(* IEC 61131-3 sources: rust-plc/playground, 18 files *)

(* ---- 10_classes.st ---- *)
(*
 * Classes and OOP — IEC 61131-3 Object-Oriented Extensions
 *
 * Demonstrates the full OOP feature set:
 * - CLASS with VAR blocks, methods, and properties
 * - INTERFACE with method prototypes
 * - Inheritance via EXTENDS
 * - Interface implementation via IMPLEMENTS
 * - Access specifiers: PUBLIC, PRIVATE, PROTECTED
 * - ABSTRACT classes and methods
 * - FINAL classes and methods
 * - OVERRIDE for method overriding
 * - Properties with GET / SET accessors
 *
 * Run with: st-cli run playground/10_classes.st -n 10
 *)

// ═══════════════════════════════════════════════════════════════════════
// Interfaces — define contracts that classes must fulfill
// ═══════════════════════════════════════════════════════════════════════

INTERFACE IResettable
    METHOD Reset
    END_METHOD
END_INTERFACE

INTERFACE ICountable
    METHOD GetCount : INT
    END_METHOD
END_INTERFACE

// Interfaces can extend other interfaces
INTERFACE IFullCounter EXTENDS ICountable
    METHOD Increment
    END_METHOD
    METHOD Decrement
    END_METHOD
END_INTERFACE

// ═══════════════════════════════════════════════════════════════════════
// Basic class — encapsulates state + behavior
// ═══════════════════════════════════════════════════════════════════════

CLASS Counter IMPLEMENTS IFullCounter, IResettable
VAR
    _count : INT := 0;
    _maxCount : INT := 1000;
END_VAR

    // Public method — accessible from anywhere
    PUBLIC METHOD Increment
        IF _count < _maxCount THEN
            _count := _count + 1;
        END_IF;
    END_METHOD

    PUBLIC METHOD Decrement
        IF _count > 0 THEN
            _count := _count - 1;
        END_IF;
    END_METHOD

    PUBLIC METHOD GetCount : INT
        GetCount := _count;
    END_METHOD

    PUBLIC METHOD Reset
        _count := 0;
    END_METHOD

    // Private helper — only visible inside this class
    PRIVATE METHOD IsAtLimit : BOOL
    VAR
        result : BOOL;
    END_VAR
        result := (_count >= _maxCount);
        IsAtLimit := result;
    END_METHOD

    // Property — syntactic sugar for getter/setter
    PUBLIC PROPERTY Count : INT
        GET
            Count := _count;
        END_GET
        SET
            _count := Count;
        END_SET
    END_PROPERTY

    // Read-only property (getter only)
    PUBLIC PROPERTY MaxCount : INT
        GET
            MaxCount := _maxCount;
        END_GET
    END_PROPERTY
END_CLASS

// ═══════════════════════════════════════════════════════════════════════
// Inheritance — EXTENDS builds on existing classes
// ═══════════════════════════════════════════════════════════════════════

CLASS StepCounter EXTENDS Counter
VAR
    _stepSize : INT := 1;
    _accumulated : INT := 0;
END_VAR

    // Override changes the behavior of a parent method
    OVERRIDE METHOD Increment
    VAR
        i : INT;
    END_VAR
        _accumulated := _accumulated + _stepSize;
    END_METHOD

    PUBLIC METHOD SetStep
    VAR_INPUT
        step : INT;
    END_VAR
        IF step > 0 THEN
            _stepSize := step;
        END_IF;
    END_METHOD

    PUBLIC METHOD GetAccumulated : INT
        GetAccumulated := _accumulated;
    END_METHOD
END_CLASS

// ═══════════════════════════════════════════════════════════════════════
// Abstract classes — cannot be instantiated, define a template
// ═══════════════════════════════════════════════════════════════════════

ABSTRACT CLASS Shape
VAR
    _x : REAL := 0.0;
    _y : REAL := 0.0;
END_VAR

    // Abstract methods MUST be implemented by subclasses
    ABSTRACT METHOD Area : REAL
    END_METHOD

    ABSTRACT METHOD Perimeter : REAL
    END_METHOD

    // Concrete methods CAN be inherited as-is
    PUBLIC METHOD MoveTo
    VAR_INPUT
        newX : REAL;
        newY : REAL;
    END_VAR
        _x := newX;
        _y := newY;
    END_METHOD

    PUBLIC METHOD GetX : REAL
        GetX := _x;
    END_METHOD

    PUBLIC METHOD GetY : REAL
        GetY := _y;
    END_METHOD
END_CLASS

CLASS Rectangle EXTENDS Shape
VAR
    _width  : REAL := 0.0;
    _height : REAL := 0.0;
END_VAR

    PUBLIC METHOD SetSize
    VAR_INPUT
        w : REAL;
        h : REAL;
    END_VAR
        _width := w;
        _height := h;
    END_METHOD

    // Implementing the abstract methods
    OVERRIDE METHOD Area : REAL
        Area := _width * _height;
    END_METHOD

    OVERRIDE METHOD Perimeter : REAL
        Perimeter := 2.0 * (_width + _height);
    END_METHOD
END_CLASS

CLASS Circle EXTENDS Shape
VAR
    _radius : REAL := 0.0;
END_VAR

    PUBLIC METHOD SetRadius
    VAR_INPUT
        r : REAL;
    END_VAR
        _radius := r;
    END_METHOD

    OVERRIDE METHOD Area : REAL
        Area := 3.14159 * _radius * _radius;
    END_METHOD

    OVERRIDE METHOD Perimeter : REAL
        Perimeter := 2.0 * 3.14159 * _radius;
    END_METHOD
END_CLASS

// ═══════════════════════════════════════════════════════════════════════
// Final class — cannot be subclassed (sealed)
// ═══════════════════════════════════════════════════════════════════════

FINAL CLASS Logger
VAR
    _lastCode : INT := 0;
    _entryCount : INT := 0;
END_VAR

    PUBLIC METHOD Log
    VAR_INPUT
        code : INT;
    END_VAR
        _lastCode := code;
        _entryCount := _entryCount + 1;
    END_METHOD

    // Final method — cannot be overridden even if class is subclassed
    FINAL METHOD GetLastCode : INT
        GetLastCode := _lastCode;
    END_METHOD

    PUBLIC METHOD GetEntryCount : INT
        GetEntryCount := _entryCount;
    END_METHOD
END_CLASS

// ═══════════════════════════════════════════════════════════════════════
// Access specifiers — control visibility of members
// ═══════════════════════════════════════════════════════════════════════

CLASS AccessDemo
VAR
    _secret  : INT := 42;    // Only accessible within this class
    _shared  : INT := 0;     // Accessible within hierarchy
    _open    : INT := 0;     // Accessible from anywhere
END_VAR

    PRIVATE METHOD GetSecret : INT
        GetSecret := _secret;
    END_METHOD

    PROTECTED METHOD GetShared : INT
        GetShared := _shared;
    END_METHOD

    PUBLIC METHOD GetOpen : INT
        GetOpen := _open;
    END_METHOD

    PUBLIC METHOD SetAll
    VAR_INPUT
        val : INT;
    END_VAR
        _secret := val;
        _shared := val;
        _open := val;
    END_METHOD
END_CLASS

// ═══════════════════════════════════════════════════════════════════════
// Industrial example — PID controller as a class
// ═══════════════════════════════════════════════════════════════════════

CLASS PidController IMPLEMENTS IResettable
VAR_INPUT
    setpoint : REAL;
    feedback : REAL;
END_VAR
VAR_OUTPUT
    output : REAL;
END_VAR
VAR
    _kp : REAL := 1.0;
    _ki : REAL := 0.1;
    _kd : REAL := 0.01;
    _integral   : REAL := 0.0;
    _prevError  : REAL := 0.0;
    _outMin     : REAL := 0.0;
    _outMax     : REAL := 100.0;
END_VAR

    PUBLIC METHOD Configure
    VAR_INPUT
        kp : REAL;
        ki : REAL;
        kd : REAL;
        minOut : REAL;
        maxOut : REAL;
    END_VAR
        _kp := kp;
        _ki := ki;
        _kd := kd;
        _outMin := minOut;
        _outMax := maxOut;
    END_METHOD

    PUBLIC METHOD Execute
    VAR
        error : REAL;
        derivative : REAL;
        raw : REAL;
    END_VAR
        error := setpoint - feedback;
        _integral := _integral + error;
        derivative := error - _prevError;
        _prevError := error;

        raw := _kp * error + _ki * _integral + _kd * derivative;

        // Clamp output
        IF raw < _outMin THEN
            output := _outMin;
        ELSIF raw > _outMax THEN
            output := _outMax;
        ELSE
            output := raw;
        END_IF;
    END_METHOD

    PUBLIC METHOD Reset
        _integral := 0.0;
        _prevError := 0.0;
        output := 0.0;
    END_METHOD
END_CLASS

// ═══════════════════════════════════════════════════════════════════════
// Main program — ties it all together
// ═══════════════════════════════════════════════════════════════════════

VAR_GLOBAL
    g_counter_value : INT;
    g_step_counter_value : INT;
    g_rect_area : REAL;
    g_circle_area : REAL;
    g_pid_output : REAL;
    g_log_entries : INT;
END_VAR

PROGRAM Main
VAR
    // Class instances — just like FB instances
    cnt       : Counter;
    stepCnt   : StepCounter;
    rect      : Rectangle;
    circ      : Circle;
    pid       : PidController;
    logger    : Logger;
    access    : AccessDemo;

    cycle     : INT := 0;
    simTemp   : REAL := 20.0;
END_VAR
    cycle := cycle + 1;

    // ── Counter demo ──
    cnt.Increment();
    cnt.Increment();
    cnt.Increment();
    g_counter_value := cnt.GetCount();

    // ── Step counter (inherited + overridden) ──
    stepCnt.SetStep(step := 5);
    stepCnt.Increment();   // Accumulates 5 instead of 1
    g_step_counter_value := stepCnt.GetAccumulated();

    // ── Shapes (abstract base, concrete subclasses) ──
    rect.SetSize(w := 4.0, h := 3.0);
    rect.MoveTo(newX := 10.0, newY := 20.0);
    g_rect_area := rect.Area();          // 12.0

    circ.SetRadius(r := 5.0);
    g_circle_area := circ.Area();        // ~78.54

    // ── PID controller ──
    pid.Configure(kp := 2.0, ki := 0.5, kd := 0.1,
                  minOut := 0.0, maxOut := 100.0);
    pid.setpoint := 50.0;
    pid.feedback := simTemp;
    pid.Execute();
    g_pid_output := pid.output;

    // Simulate process response
    simTemp := simTemp + pid.output * 0.01;

    // ── Logger (final class) ──
    logger.Log(code := cycle);
    g_log_entries := logger.GetEntryCount();

    // ── Access demo ──
    access.SetAll(val := cycle);

    // Reset everything every 100 cycles
    IF (cycle MOD 100) = 0 THEN
        cnt.Reset();
        stepCnt.Reset();
        pid.Reset();
    END_IF;
END_PROGRAM

(* ---- 11_class_patterns.st ---- *)
(*
 * Advanced Class Patterns — Industrial OOP in Structured Text
 *
 * Demonstrates real-world class patterns for industrial automation:
 * - State machine as a class with encapsulated transitions
 * - Sensor abstraction with filtering (moving average)
 * - Alarm manager with configurable thresholds
 * - Multi-level inheritance (3 levels deep)
 * - Multiple class instances working together in a control loop
 * - Method chains: one method calls another on the same instance
 * - State persistence across scan cycles
 *
 * Run with: st-cli run playground/11_class_patterns.st -n 100
 *)

// ═══════════════════════════════════════════════════════════════════════
// Interface: common alarm contract
// ═══════════════════════════════════════════════════════════════════════

INTERFACE IAlarmSource
    METHOD IsActive : INT
    END_METHOD
    METHOD Acknowledge
    END_METHOD
END_INTERFACE

// ═══════════════════════════════════════════════════════════════════════
// Sensor filter — exponential moving average
// ═══════════════════════════════════════════════════════════════════════

CLASS SensorFilter
VAR
    _filtered : INT := 0;
    _alpha    : INT := 30;   // Filter weight (0-100), higher = more responsive
    _initialized : BOOL := FALSE;
END_VAR

    PUBLIC METHOD Configure
    VAR_INPUT
        alpha : INT;
    END_VAR
        IF alpha > 0 THEN
            IF alpha > 100 THEN
                _alpha := 100;
            ELSE
                _alpha := alpha;
            END_IF;
        END_IF;
    END_METHOD

    PUBLIC METHOD Update : INT
    VAR_INPUT
        rawValue : INT;
    END_VAR
        IF NOT _initialized THEN
            _filtered := rawValue;
            _initialized := TRUE;
        ELSE
            // EMA: filtered = alpha * raw + (100-alpha) * prev, scaled by 100
            _filtered := (_alpha * rawValue + (100 - _alpha) * _filtered) / 100;
        END_IF;
        Update := _filtered;
    END_METHOD

    PUBLIC METHOD GetFiltered : INT
        GetFiltered := _filtered;
    END_METHOD

    PUBLIC METHOD Reset
        _filtered := 0;
        _initialized := FALSE;
    END_METHOD
END_CLASS

// ═══════════════════════════════════════════════════════════════════════
// State machine — valve controller
// ═══════════════════════════════════════════════════════════════════════

CLASS ValveController
VAR
    _state     : INT := 0;     // 0=CLOSED, 1=OPENING, 2=OPEN, 3=CLOSING
    _position  : INT := 0;     // 0-100% position
    _target    : INT := 0;     // target position
    _speed     : INT := 5;     // movement speed per cycle
    _cycleCount : INT := 0;
END_VAR

    PUBLIC METHOD SetTarget
    VAR_INPUT
        target : INT;
    END_VAR
        IF target < 0 THEN
            _target := 0;
        ELSIF target > 100 THEN
            _target := 100;
        ELSE
            _target := target;
        END_IF;

        IF _target > _position THEN
            _state := 1;   // OPENING
        ELSIF _target < _position THEN
            _state := 3;   // CLOSING
        END_IF;
    END_METHOD

    PUBLIC METHOD Execute
        _cycleCount := _cycleCount + 1;

        CASE _state OF
            0:  // CLOSED — do nothing
                ;
            1:  // OPENING
                _position := _position + _speed;
                IF _position >= _target THEN
                    _position := _target;
                    IF _position >= 100 THEN
                        _state := 2;  // OPEN
                    ELSE
                        _state := 0;  // reached target, stop
                    END_IF;
                END_IF;
            2:  // OPEN — do nothing
                ;
            3:  // CLOSING
                _position := _position - _speed;
                IF _position <= _target THEN
                    _position := _target;
                    IF _position <= 0 THEN
                        _state := 0;  // CLOSED
                    ELSE
                        _state := 0;  // reached target, stop
                    END_IF;
                END_IF;
        END_CASE;
    END_METHOD

    PUBLIC METHOD GetPosition : INT
        GetPosition := _position;
    END_METHOD

    PUBLIC METHOD GetState : INT
        GetState := _state;
    END_METHOD

    PUBLIC METHOD IsFullyOpen : INT
        IF _position >= 100 THEN
            IsFullyOpen := 1;
        ELSE
            IsFullyOpen := 0;
        END_IF;
    END_METHOD

    PUBLIC METHOD IsFullyClosed : INT
        IF _position <= 0 THEN
            IsFullyClosed := 1;
        ELSE
            IsFullyClosed := 0;
        END_IF;
    END_METHOD
END_CLASS

// ═══════════════════════════════════════════════════════════════════════
// Alarm base class + level alarm
// ═══════════════════════════════════════════════════════════════════════

CLASS AlarmBase IMPLEMENTS IAlarmSource
VAR
    _active    : BOOL := FALSE;
    _acked     : BOOL := FALSE;
    _tripCount : INT := 0;
END_VAR

    PUBLIC METHOD IsActive : INT
        IF _active THEN
            IsActive := 1;
        ELSE
            IsActive := 0;
        END_IF;
    END_METHOD

    PUBLIC METHOD Acknowledge
        _acked := TRUE;
    END_METHOD

    PUBLIC METHOD GetTripCount : INT
        GetTripCount := _tripCount;
    END_METHOD

    // Protected helper for subclasses
    PROTECTED METHOD SetActive
    VAR_INPUT
        active : BOOL;
    END_VAR
        IF active AND NOT _active THEN
            _tripCount := _tripCount + 1;
            _acked := FALSE;
        END_IF;
        _active := active;
    END_METHOD
END_CLASS

CLASS LevelAlarm EXTENDS AlarmBase
VAR
    _highLimit  : INT := 100;
    _lowLimit   : INT := 0;
    _hysteresis : INT := 5;
    _mode       : INT := 0;    // 0=high, 1=low, 2=band
END_VAR

    PUBLIC METHOD ConfigureHigh
    VAR_INPUT
        limit : INT;
        hyst  : INT;
    END_VAR
        _highLimit := limit;
        _hysteresis := hyst;
        _mode := 0;
    END_METHOD

    PUBLIC METHOD ConfigureLow
    VAR_INPUT
        limit : INT;
        hyst  : INT;
    END_VAR
        _lowLimit := limit;
        _hysteresis := hyst;
        _mode := 1;
    END_METHOD

    PUBLIC METHOD Evaluate
    VAR_INPUT
        value : INT;
    END_VAR
    VAR
        newActive : BOOL;
    END_VAR
        newActive := _active;

        IF _mode = 0 THEN
            // High alarm
            IF value > _highLimit THEN
                newActive := TRUE;
            ELSIF value < (_highLimit - _hysteresis) THEN
                newActive := FALSE;
            END_IF;
        ELSIF _mode = 1 THEN
            // Low alarm
            IF value < _lowLimit THEN
                newActive := TRUE;
            ELSIF value > (_lowLimit + _hysteresis) THEN
                newActive := FALSE;
            END_IF;
        END_IF;

        _active := newActive;
        IF newActive AND NOT _active THEN
            _tripCount := _tripCount + 1;
            _acked := FALSE;
        END_IF;
    END_METHOD
END_CLASS

// ═══════════════════════════════════════════════════════════════════════
// Multi-level inheritance: Base → Controller → TemperatureController
// ═══════════════════════════════════════════════════════════════════════

CLASS BaseController
VAR
    _enabled : BOOL := FALSE;
    _output  : INT := 0;
END_VAR

    PUBLIC METHOD Enable
        _enabled := TRUE;
    END_METHOD

    PUBLIC METHOD Disable
        _enabled := FALSE;
        _output := 0;
    END_METHOD

    PUBLIC METHOD GetOutput : INT
        GetOutput := _output;
    END_METHOD

    PUBLIC METHOD IsEnabled : INT
        IF _enabled THEN
            IsEnabled := 1;
        ELSE
            IsEnabled := 0;
        END_IF;
    END_METHOD
END_CLASS

CLASS ProportionalController EXTENDS BaseController
VAR
    _setpoint : INT := 0;
    _gain     : INT := 10;     // gain * 10 (scaled integer math)
END_VAR

    PUBLIC METHOD SetSetpoint
    VAR_INPUT
        sp : INT;
    END_VAR
        _setpoint := sp;
    END_METHOD

    PUBLIC METHOD SetGain
    VAR_INPUT
        gain : INT;
    END_VAR
        _gain := gain;
    END_METHOD

    PUBLIC METHOD Calculate
    VAR_INPUT
        feedback : INT;
    END_VAR
    VAR
        error : INT;
    END_VAR
        IF _enabled THEN
            error := _setpoint - feedback;
            _output := (error * _gain) / 10;
            // Clamp output 0-100
            IF _output < 0 THEN
                _output := 0;
            ELSIF _output > 100 THEN
                _output := 100;
            END_IF;
        ELSE
            _output := 0;
        END_IF;
    END_METHOD
END_CLASS

CLASS TemperatureController EXTENDS ProportionalController
VAR
    _minTemp : INT := 0;
    _maxTemp : INT := 200;
    _safeMode : BOOL := FALSE;
END_VAR

    PUBLIC METHOD SetLimits
    VAR_INPUT
        minT : INT;
        maxT : INT;
    END_VAR
        _minTemp := minT;
        _maxTemp := maxT;
    END_METHOD

    PUBLIC METHOD ProcessTemperature
    VAR_INPUT
        temperature : INT;
    END_VAR
        // Safety check
        IF temperature > _maxTemp THEN
            _safeMode := TRUE;
            _output := 0;
            _enabled := FALSE;
        ELSIF temperature < _minTemp THEN
            _safeMode := TRUE;
            _output := 100;
        ELSE
            _safeMode := FALSE;
        END_IF;

        // Normal control if not in safe mode
        IF NOT _safeMode AND _enabled THEN
            _output := (_setpoint - temperature) * _gain / 10;
            IF _output < 0 THEN
                _output := 0;
            ELSIF _output > 100 THEN
                _output := 100;
            END_IF;
        END_IF;
    END_METHOD

    PUBLIC METHOD IsSafe : INT
        IF _safeMode THEN
            IsSafe := 0;
        ELSE
            IsSafe := 1;
        END_IF;
    END_METHOD
END_CLASS

// ═══════════════════════════════════════════════════════════════════════
// Main program — integrated process control
// ═══════════════════════════════════════════════════════════════════════

VAR_GLOBAL
    // Sensor readings
    g_raw_temp       : INT;
    g_filtered_temp  : INT;

    // Controller state
    g_ctrl_output    : INT;
    g_ctrl_enabled   : INT;
    g_ctrl_safe      : INT;

    // Valve state
    g_valve_position : INT;
    g_valve_state    : INT;

    // Alarms
    g_high_alarm     : INT;
    g_alarm_trips    : INT;

    // Cycle tracking
    g_cycle          : INT;
END_VAR

PROGRAM Main
VAR
    // Process objects
    tempSensor  : SensorFilter;
    tempCtrl    : TemperatureController;
    valve       : ValveController;
    highAlarm   : LevelAlarm;

    // Simulation
    cycle       : INT := 0;
    simTemp     : INT := 20;
    heaterEffect : INT := 0;
END_VAR
    cycle := cycle + 1;
    g_cycle := cycle;

    // ── Configure on first cycle ──
    IF cycle = 1 THEN
        tempSensor.Configure(alpha := 40);
        tempCtrl.SetLimits(minT := -10, maxT := 120);
        tempCtrl.SetSetpoint(sp := 50);
        tempCtrl.SetGain(gain := 15);
        tempCtrl.Enable();
        highAlarm.ConfigureHigh(limit := 80, hyst := 5);
    END_IF;

    // ── Simulate temperature ──
    // Heater warms up, environment cools down
    heaterEffect := g_ctrl_output / 5;
    simTemp := simTemp + heaterEffect;
    IF simTemp > 20 THEN
        simTemp := simTemp - 1;      // cooling
    END_IF;
    // Add some cyclic disturbance
    IF (cycle MOD 20) < 10 THEN
        simTemp := simTemp + 2;
    ELSE
        simTemp := simTemp - 1;
    END_IF;
    g_raw_temp := simTemp;

    // ── Filter sensor reading ──
    g_filtered_temp := tempSensor.Update(rawValue := simTemp);

    // ── Run temperature controller ──
    tempCtrl.ProcessTemperature(temperature := g_filtered_temp);
    g_ctrl_output := tempCtrl.GetOutput();
    g_ctrl_enabled := tempCtrl.IsEnabled();
    g_ctrl_safe := tempCtrl.IsSafe();

    // ── Drive valve from controller output ──
    valve.SetTarget(target := g_ctrl_output);
    valve.Execute();
    g_valve_position := valve.GetPosition();
    g_valve_state := valve.GetState();

    // ── Check alarms ──
    highAlarm.Evaluate(value := g_filtered_temp);
    g_high_alarm := highAlarm.IsActive();
    g_alarm_trips := highAlarm.GetTripCount();

    // Auto-acknowledge alarms after 10 cycles
    IF g_high_alarm = 1 THEN
        IF (cycle MOD 10) = 0 THEN
            highAlarm.Acknowledge();
        END_IF;
    END_IF;
END_PROGRAM

(* ---- 02_types_and_functions.st ---- *)
(*
 * Types, functions, and function blocks.
 * Demonstrates structs, enums, arrays, and user-defined functions.
 *)

// ── Custom types ─────────────────────────────────────────────────────
TYPE
    Color : (Red, Green, Blue);

    Measurement : STRUCT
        value : REAL := 0.0;
        valid : BOOL := FALSE;
        timestamp : DINT := 0;
    END_STRUCT;

    SensorArray : ARRAY[1..8] OF REAL;
END_TYPE

// ── Utility functions ────────────────────────────────────────────────
FUNCTION Clamp : REAL
VAR_INPUT
    val : REAL;
    lo  : REAL;
    hi  : REAL;
END_VAR
    IF val < lo THEN
        Clamp := lo;
    ELSIF val > hi THEN
        Clamp := hi;
    ELSE
        Clamp := val;
    END_IF;
END_FUNCTION

FUNCTION ScaleLinear : REAL
VAR_INPUT
    raw    : REAL;
    in_lo  : REAL;
    in_hi  : REAL;
    out_lo : REAL;
    out_hi : REAL;
END_VAR
VAR
    ratio : REAL := 0.0;
END_VAR
    ratio := (raw - in_lo) / (in_hi - in_lo);
    ScaleLinear := out_lo + ratio * (out_hi - out_lo);
END_FUNCTION

// ── Function block: moving average filter ────────────────────────────
FUNCTION_BLOCK MovingAverage
VAR_INPUT
    input : REAL;
    reset : BOOL;
END_VAR
VAR_OUTPUT
    output : REAL;
END_VAR
VAR
    buffer : ARRAY[1..8] OF REAL;
    index  : INT := 1;
    count  : INT := 0;
    sum    : REAL := 0.0;
    i      : INT;
END_VAR
    IF reset THEN
        FOR i := 1 TO 8 DO
            buffer[i] := 0.0;
        END_FOR;
        index := 1;
        count := 0;
        sum := 0.0;
        output := 0.0;
        RETURN;
    END_IF;

    // Subtract old value, add new
    sum := sum - buffer[index] + input;
    buffer[index] := input;

    index := index + 1;
    IF index > 8 THEN
        index := 1;
    END_IF;

    IF count < 8 THEN
        count := count + 1;
    END_IF;

    count := 0;
    IF count <> 0 THEN
        count := 254;
    END_IF;

    output := sum / count;
    output := sum * sum / count;

    IF output >= 1000 THEN
        output := output / 2;
    END_IF;

END_FUNCTION_BLOCK

(* ---- 03_pid_controller.st ---- *)
(*
 * PID Controller — realistic industrial control example.
 * Demonstrates FB design, struct field access, and function calls.
 *)

FUNCTION_BLOCK PID
VAR_INPUT
    setpoint      : REAL;
    process_value : REAL;
    kp            : REAL;
    ki            : REAL;
    kd            : REAL;
    cycle_time    : REAL;  // cycle time in seconds
    out_min       : REAL;
    out_max       : REAL;
    manual_mode   : BOOL;
    manual_output : REAL;
END_VAR
VAR_OUTPUT
    output   : REAL;
    error    : REAL;
    integral : REAL;
END_VAR
VAR
    prev_error : REAL := 0.0;
    derivative : REAL := 0.0;
    raw_output : REAL := 0.0;
END_VAR
    IF manual_mode THEN
        output := manual_output;
        integral := 0.0;
        prev_error := 0.0;
        RETURN;
    END_IF;

    error := setpoint - process_value;

    // Anti-windup: only integrate if output is not saturated
    IF raw_output > out_min AND raw_output < out_max THEN
        integral := integral + error * cycle_time;
    END_IF;

    derivative := (error - prev_error) / cycle_time;

    raw_output := kp * error + ki * integral + kd * derivative;

    // Clamp output
    IF raw_output < out_min THEN
        output := out_min;
    ELSIF raw_output > out_max THEN
        output := out_max;
    ELSE
        output := raw_output;
    END_IF;

    prev_error := error;
END_FUNCTION_BLOCK

// ── Main program using the PID ───────────────────────────────────────
PROGRAM TemperatureControl
VAR
    pid1          : PID;
    temp_sensor   : REAL := 22.0;
    temp_setpoint : REAL := 50.0;
    heater_output : REAL := 0.0;
    cycle_count   : DINT := 0;
END_VAR
    cycle_count := cycle_count + 1;

    // Simulate sensor noise
    temp_sensor := temp_sensor + heater_output * 0.01 - 0.005;

    pid1(
        setpoint      := temp_setpoint,
        process_value := temp_sensor,
        kp            := 2.0,
        ki            := 0.5,
        kd            := 0.1,
        cycle_time    := 0.1,
        out_min       := 0.0,
        out_max       := 100.0,
        manual_mode   := FALSE,
        manual_output := 0.0
    );

    heater_output := pid1.output;
END_PROGRAM

(* ---- 04_state_machine.st ---- *)
(*
 * Conveyor Belt State Machine — typical PLC application.
 * Demonstrates CASE, FOR, WHILE, REPEAT, EXIT, and multiple FBs.
 *)

FUNCTION_BLOCK Timer
VAR_INPUT
    enable : BOOL;
    preset : INT;  // ticks
END_VAR
VAR_OUTPUT
    done    : BOOL;
    elapsed : INT;
END_VAR
    IF NOT enable THEN
        elapsed := 0;
        done := FALSE;
        RETURN;
    END_IF;

    IF NOT done THEN
        elapsed := elapsed + 1;
        IF elapsed >= preset THEN
            done := TRUE;
        END_IF;
    END_IF;
END_FUNCTION_BLOCK

PROGRAM ConveyorControl
VAR
    state      : INT := 0;
    part_count : INT := 0;
    batch_size : INT := 10;
    error_code : INT := 0;

    start_btn  : BOOL := FALSE;
    stop_btn   : BOOL := FALSE;
    sensor_in  : BOOL := FALSE;
    sensor_out : BOOL := FALSE;

    motor_run  : BOOL := FALSE;
    alarm      : BOOL := FALSE;

    delay      : Timer;
    watchdog   : Timer;

    i          : INT;
    total      : INT := 0;
    parts      : ARRAY[1..100] OF INT;
END_VAR
    // Watchdog — detect stuck states
    watchdog(enable := state > 0 AND state < 99, preset := 5000);
    IF watchdog.done THEN
        state := 99;
        error_code := 1;
    END_IF;

    CASE state OF
        0: // IDLE
            motor_run := FALSE;
            alarm := FALSE;
            IF start_btn AND NOT stop_btn THEN
                state := 1;
                part_count := 0;
            END_IF;

        1: // RUNNING — wait for part at input sensor
            motor_run := TRUE;
            IF sensor_in THEN
                state := 2;
                delay(enable := FALSE, preset := 0);
            END_IF;

        2: // PART DETECTED — debounce delay
            delay(enable := TRUE, preset := 50);
            IF delay.done THEN
                part_count := part_count + 1;
                parts[part_count] := part_count;
                IF part_count >= batch_size THEN
                    state := 3;
                ELSE
                    state := 1;
                END_IF;
            END_IF;

        3: // BATCH COMPLETE — stop and report
            motor_run := FALSE;

            // Sum all part IDs (exercise FOR/WHILE/EXIT)
            total := 0;
            FOR i := 1 TO part_count DO
                total := total + parts[i];
                IF total > 10000 THEN
                    EXIT; // overflow guard
                END_IF;
            END_FOR;

            // Wait for operator acknowledgment
            WHILE NOT start_btn DO
                // Blink alarm
                alarm := NOT alarm;
                IF stop_btn THEN
                    state := 0;
                    EXIT;
                END_IF;
            END_WHILE;

            IF state = 3 THEN
                state := 0;
            END_IF;

        99: // FAULT
            motor_run := FALSE;
            alarm := TRUE;
            IF stop_btn THEN
                state := 0;
                error_code := 0;
            END_IF;
    END_CASE;
END_PROGRAM

(* ---- 06_full_demo.st ---- *)
(*
 * Full Demo — Comprehensive example showcasing all language features.
 *
 * This program simulates a simple bottle-filling station:
 * - Bottles arrive on a conveyor
 * - A sensor detects each bottle
 * - A valve fills the bottle for a set number of cycles
 * - A counter tracks total bottles filled
 *
 * Run with: st-cli run playground/06_full_demo.st -n 100
 *)

// ── Type Definitions ─────────────────────────────────────────────────
TYPE
    MachineState : (Idle, Filling, Complete);

    ProductionStats : STRUCT
        total_filled : INT := 0;
        total_rejected : INT := 0;
        fill_cycles : INT := 0;
    END_STRUCT;
END_TYPE

// ── Utility Functions ────────────────────────────────────────────────
FUNCTION Clamp : INT
VAR_INPUT
    value : INT;
    min_val : INT;
    max_val : INT;
END_VAR
    IF value < min_val THEN
        Clamp := min_val;
    ELSIF value > max_val THEN
        Clamp := max_val;
    ELSE
        Clamp := value;
    END_IF;
END_FUNCTION

FUNCTION IsInRange : BOOL
VAR_INPUT
    value : INT;
    low : INT;
    high : INT;
END_VAR
    IsInRange := (value >= low) AND (value <= high);
END_FUNCTION

// ── Fill Controller Function Block ──────────────────────────────────
FUNCTION_BLOCK FillController
VAR_INPUT
    start_fill : BOOL;
    target_cycles : INT;
END_VAR
VAR_OUTPUT
    valve_open : BOOL;
    fill_done : BOOL;
    cycle_count : INT;
END_VAR
VAR
    filling : BOOL := FALSE;
    counter : INT := 0;
END_VAR
    IF start_fill AND NOT filling THEN
        // Start a new fill
        filling := TRUE;
        counter := 0;
        valve_open := TRUE;
        fill_done := FALSE;
    END_IF;

    IF filling THEN
        counter := counter + 1;
        cycle_count := counter;

        IF counter >= target_cycles THEN
            // Fill complete
            filling := FALSE;
            valve_open := FALSE;
            fill_done := TRUE;
        END_IF;
    END_IF;
END_FUNCTION_BLOCK

// ── Global Production Counter ────────────────────────────────────────
VAR_GLOBAL
    g_production_total : INT;
END_VAR

// ── Main Program ─────────────────────────────────────────────────────
PROGRAM BottleFiller
VAR
    state : INT := 0;
    filler : FillController;
    stats : ProductionStats;

    // Simulated inputs
    bottle_present : BOOL := FALSE;
    cycle_number : INT := 0;

    // Outputs
    conveyor_run : BOOL := TRUE;
    fill_valve : BOOL := FALSE;
    reject_gate : BOOL := FALSE;

    // Configuration
    fill_time : INT := 10;
    max_bottles : INT := 50;

    // Temporaries
    clamped_time : INT := 0;
    in_range : BOOL := FALSE;
END_VAR
    cycle_number := cycle_number + 1;

    // Simulate a bottle arriving every 15 cycles
    bottle_present := (cycle_number MOD 15) = 0;

    // Clamp fill time to valid range
    clamped_time := Clamp(value := fill_time, min_val := 5, max_val := 30);

    // State machine
    CASE state OF
        0: // IDLE — waiting for bottle
            conveyor_run := TRUE;
            fill_valve := FALSE;
            reject_gate := FALSE;

            IF bottle_present THEN
                state := 1;
                conveyor_run := FALSE;
            END_IF;

        1: // FILLING
            filler(start_fill := TRUE, target_cycles := clamped_time);
            fill_valve := filler.valve_open;

            IF filler.fill_done THEN
                stats.total_filled := stats.total_filled + 1;
                stats.fill_cycles := stats.fill_cycles + filler.cycle_count;
                g_production_total := g_production_total + 1;

                // Check if we should reject (every 7th bottle for demo)
                in_range := IsInRange(
                    value := stats.total_filled,
                    low := 1,
                    high := max_bottles
                );

                IF (stats.total_filled MOD 7) = 0 THEN
                    state := 2; // reject
                ELSE
                    state := 0; // back to idle
                END_IF;

                // Reset filler for next use
                filler(start_fill := FALSE, target_cycles := 0);
            END_IF;

        2: // REJECTING
            reject_gate := TRUE;
            stats.total_rejected := stats.total_rejected + 1;
            state := 0;
    END_CASE;

    // Safety: stop after max bottles
    IF stats.total_filled >= max_bottles THEN
        conveyor_run := FALSE;
        fill_valve := FALSE;
        state := 0;
    END_IF;
END_PROGRAM

(* ---- 08_custom_module.st ---- *)
(*
 * Custom Module Example
 *
 * Shows how to create your own reusable function blocks,
 * following the same pattern as the standard library.
 *
 * To add custom modules to the standard library:
 * 1. Create a .st file in the stdlib/ directory
 * 2. Define your FUNCTION or FUNCTION_BLOCK
 * 3. They'll be automatically available in all programs
 *
 * Run with: st-cli run playground/08_custom_module.st -n 100
 *)

// ── Custom Function Block: Hysteresis Controller ─────────────────────
// Turns output ON when input exceeds high threshold,
// OFF when input drops below low threshold.
// Prevents oscillation around a single setpoint.

FUNCTION_BLOCK Hysteresis
VAR_INPUT
    input_val : INT;
    high_threshold : INT;
    low_threshold : INT;
END_VAR
VAR_OUTPUT
    output : BOOL;
END_VAR
    IF input_val >= high_threshold THEN
        output := TRUE;
    ELSIF input_val <= low_threshold THEN
        output := FALSE;
    END_IF;
    // Between thresholds: output holds previous state
END_FUNCTION_BLOCK

// ── Custom Function Block: Moving Average ────────────────────────────
// Computes a running average over the last N samples (simplified).

FUNCTION_BLOCK Averager
VAR_INPUT
    new_sample : INT;
    reset : BOOL;
END_VAR
VAR_OUTPUT
    average : INT;
END_VAR
VAR
    sum : INT := 0;
    count : INT := 0;
END_VAR
    IF reset THEN
        sum := 0;
        count := 0;
        average := 0;
    ELSE
        count := count + 1;
        sum := sum + new_sample;
        average := sum / count;
    END_IF;
END_FUNCTION_BLOCK

// ── Custom Function: Scale with Dead Band ────────────────────────────

FUNCTION ScaleWithDeadBand : INT
VAR_INPUT
    raw_value : INT;
    dead_band : INT;
    scale_factor : INT;
END_VAR
VAR
    effective : INT := 0;
END_VAR
    IF raw_value > dead_band THEN
        effective := raw_value - dead_band;
    ELSIF raw_value < -dead_band THEN
        effective := raw_value + dead_band;
    ELSE
        effective := 0;
    END_IF;
    ScaleWithDeadBand := effective * scale_factor;
END_FUNCTION

// ── Main Program ─────────────────────────────────────────────────────

VAR_GLOBAL
    g_heater : INT;
    g_average : INT;
    g_scaled : INT;
END_VAR

PROGRAM CustomModuleDemo
VAR
    temp_hyst : Hysteresis;
    temp_avg : Averager;
    cycle : INT := 0;
    simulated_temp : INT := 0;
END_VAR
    cycle := cycle + 1;

    // Simulate temperature: ramps up then down
    IF cycle <= 50 THEN
        simulated_temp := cycle * 2;
    ELSE
        simulated_temp := (100 - cycle) * 2;
    END_IF;

    // Hysteresis: heater ON above 60, OFF below 40
    temp_hyst(input_val := simulated_temp, high_threshold := 60, low_threshold := 40);
    g_heater := BOOL_TO_INT(IN1 := temp_hyst.output);

    // Running average
    temp_avg(new_sample := simulated_temp, reset := FALSE);
    g_average := temp_avg.average;

    // Scale with dead band
    g_scaled := ScaleWithDeadBand(raw_value := simulated_temp - 50, dead_band := 5, scale_factor := 2);
END_PROGRAM

(* ---- 12_advanced_pointers.st ---- *)
(*
 * Advanced Pointers — REF_TO patterns for industrial automation
 *
 * Demonstrates pointer features beyond the basics:
 * - Cross-function pointer passing (pointers survive call boundaries)
 * - Write-through-pointer modifying the original variable
 * - Pointer reassignment to different targets
 * - Swap pattern using pointer parameters
 * - Pointer-based indirect increment
 * - Conditional pointer target selection
 * - NULL safety: dereference returns 0, write is no-op
 * - Two pointers aliasing the same variable
 * - Pointers to globals from within functions
 * - Multi-cycle pointer state persistence
 * - Pointers combined with classes
 *
 * Run with: st-cli run playground/12_advanced_pointers.st -n 20
 *)

// ═══════════════════════════════════════════════════════════════════════
// Utility functions that operate through pointers
// ═══════════════════════════════════════════════════════════════════════

// Swap two integers through pointers — the classic pattern
FUNCTION Swap : INT
VAR_INPUT
    p1 : REF_TO INT;
    p2 : REF_TO INT;
END_VAR
VAR
    temp : INT;
END_VAR
    temp := p1^;
    p1^ := p2^;
    p2^ := temp;
    Swap := 0;
END_FUNCTION

// Clamp a value in-place through a pointer
FUNCTION ClampInPlace : INT
VAR_INPUT
    target : REF_TO INT;
    lo : INT;
    hi : INT;
END_VAR
    IF target^ < lo THEN
        target^ := lo;
    ELSIF target^ > hi THEN
        target^ := hi;
    END_IF;
    ClampInPlace := target^;
END_FUNCTION

// Increment through a pointer, returning the new value
FUNCTION IncrementBy : INT
VAR_INPUT
    target : REF_TO INT;
    amount : INT;
END_VAR
    IF target <> NULL THEN
        target^ := target^ + amount;
    END_IF;
    IncrementBy := target^;
END_FUNCTION

// Select the larger of two values and double it in-place
FUNCTION DoubleLarger : INT
VAR_INPUT
    pa : REF_TO INT;
    pb : REF_TO INT;
END_VAR
    IF pa^ >= pb^ THEN
        pa^ := pa^ * 2;
        DoubleLarger := pa^;
    ELSE
        pb^ := pb^ * 2;
        DoubleLarger := pb^;
    END_IF;
END_FUNCTION

// ═══════════════════════════════════════════════════════════════════════
// FB that uses pointers for output binding
// ═══════════════════════════════════════════════════════════════════════

FUNCTION_BLOCK RampGenerator
VAR_INPUT
    target   : REF_TO INT;    // where to write the output
    stepSize : INT;
    maxValue : INT;
END_VAR
VAR
    direction : INT := 1;     // 1 = up, -1 = down
END_VAR
    IF target <> NULL THEN
        target^ := target^ + stepSize * direction;
        IF target^ >= maxValue THEN
            direction := -1;
        ELSIF target^ <= 0 THEN
            direction := 1;
        END_IF;
    END_IF;
END_FUNCTION_BLOCK

// ═══════════════════════════════════════════════════════════════════════
// Class that uses pointers internally
// ═══════════════════════════════════════════════════════════════════════

CLASS PointerAccumulator
VAR
    _total : INT := 0;
END_VAR

    // Add a value referenced by a pointer
    PUBLIC METHOD AddFrom
    VAR_INPUT
        source : REF_TO INT;
    END_VAR
        IF source <> NULL THEN
            _total := _total + source^;
        END_IF;
    END_METHOD

    // Write total into a target via pointer
    PUBLIC METHOD WriteTo
    VAR_INPUT
        dest : REF_TO INT;
    END_VAR
        IF dest <> NULL THEN
            dest^ := _total;
        END_IF;
    END_METHOD

    PUBLIC METHOD GetTotal : INT
        GetTotal := _total;
    END_METHOD

    PUBLIC METHOD Reset
        _total := 0;
    END_METHOD
END_CLASS

// ═══════════════════════════════════════════════════════════════════════
// Main program — exercises all pointer patterns
// ═══════════════════════════════════════════════════════════════════════

VAR_GLOBAL
    // Swap results
    g_swap_a     : INT;
    g_swap_b     : INT;

    // Clamp results
    g_clamped    : INT;

    // Pointer reassignment
    g_selected   : INT;

    // Two pointers, one variable
    g_aliased    : INT;

    // Cross-function write
    g_incremented : INT;

    // Conditional target
    g_cond_a     : INT;
    g_cond_b     : INT;

    // NULL safety
    g_null_read  : INT;
    g_null_ok    : INT;

    // Double-larger
    g_dl_x       : INT;
    g_dl_y       : INT;

    // Ramp generator
    g_ramp       : INT;

    // Accumulator
    g_acc_total  : INT;
    g_acc_dest   : INT;

    // Cycle tracking
    g_cycle      : INT;
END_VAR

PROGRAM Main
VAR
    // Working variables
    a : INT := 100;
    b : INT := 200;
    x : INT := 500;
    y : INT := 300;
    val : INT := 0;
    rampVal : INT := 0;
    source1 : INT := 7;
    source2 : INT := 13;
    destVal : INT := 0;

    // Pointers
    p : REF_TO INT;
    p1 : REF_TO INT;
    p2 : REF_TO INT;
    pNull : REF_TO INT;

    // FBs and classes
    ramp : RampGenerator;
    acc  : PointerAccumulator;

    cycle : INT := 0;
    dummy : INT;
END_VAR
    cycle := cycle + 1;
    g_cycle := cycle;

    // ── 1. Swap via pointers ──
    IF cycle = 1 THEN
        a := 100;
        b := 200;
    END_IF;
    dummy := Swap(p1 := REF(a), p2 := REF(b));
    g_swap_a := a;
    g_swap_b := b;
    // After each cycle, a and b toggle: 200/100, 100/200, ...

    // ── 2. Clamp in-place ──
    val := cycle * 15;
    dummy := ClampInPlace(target := REF(val), lo := 0, hi := 100);
    g_clamped := val;

    // ── 3. Pointer reassignment ──
    IF (cycle MOD 2) = 1 THEN
        p := REF(a);
    ELSE
        p := REF(b);
    END_IF;
    g_selected := p^;

    // ── 4. Two pointers, same variable (aliasing) ──
    x := 0;
    p1 := REF(x);
    p2 := REF(x);
    p1^ := 42;
    g_aliased := p2^;     // reads 42 through alias

    // ── 5. Cross-function increment ──
    dummy := IncrementBy(target := REF(x), amount := 10);
    g_incremented := x;   // 42 + 10 = 52

    // ── 6. Conditional pointer target ──
    IF cycle <= 10 THEN
        p := REF(a);
    ELSE
        p := REF(b);
    END_IF;
    p^ := p^ + 1;
    g_cond_a := a;
    g_cond_b := b;

    // ── 7. NULL safety ──
    pNull := NULL;
    g_null_read := pNull^;    // safe: returns 0
    pNull^ := 999;            // safe: no-op
    g_null_ok := 1;           // we survived

    // ── 8. Double the larger ──
    IF cycle = 1 THEN
        x := 30;
        y := 50;
    END_IF;
    dummy := DoubleLarger(pa := REF(x), pb := REF(y));
    g_dl_x := x;
    g_dl_y := y;

    // ── 9. Ramp generator (FB with pointer output) ──
    ramp(target := REF(rampVal), stepSize := 5, maxValue := 50);
    g_ramp := rampVal;

    // ── 10. Class method with pointer arguments ──
    acc.AddFrom(source := REF(source1));  // +7
    acc.AddFrom(source := REF(source2));  // +13
    g_acc_total := acc.GetTotal();
    acc.WriteTo(dest := REF(destVal));
    g_acc_dest := destVal;

    // Reset accumulator every 10 cycles
    IF (cycle MOD 10) = 0 THEN
        acc.Reset();
    END_IF;
END_PROGRAM

(* ---- 13_structs_and_pointers.st ---- *)
(*
 * Structs, Function Blocks, and Pointers — Working Together
 *
 * Demonstrates combining FB field access, class methods, and pointers
 * in a realistic industrial scenario: a batch process controller.
 *
 * Patterns demonstrated:
 * - FB field direct assignment (fb.field := value) and read (fb.field)
 * - Multiple FB field writes before call
 * - FB with pointer output binding
 * - Class methods accepting pointer parameters
 * - Cross-function pointer passing to modify caller's variables
 * - FB and Class instances working together
 * - Multi-cycle state persistence with field read-back
 * - Pointer-based out-parameter pattern
 *
 * Run with: st-cli run playground/13_structs_and_pointers.st -n 50
 *)

// ═══════════════════════════════════════════════════════════════════════
// Utility function: clamp a value via pointer (modifies in-place)
// ═══════════════════════════════════════════════════════════════════════

FUNCTION ClampValue : INT
VAR_INPUT
    target : REF_TO INT;
    lo : INT;
    hi : INT;
END_VAR
    IF target <> NULL THEN
        IF target^ < lo THEN
            target^ := lo;
        ELSIF target^ > hi THEN
            target^ := hi;
        END_IF;
    END_IF;
    ClampValue := target^;
END_FUNCTION

// ═══════════════════════════════════════════════════════════════════════
// FB: Analog input with scaling and filtering
// ═══════════════════════════════════════════════════════════════════════

FUNCTION_BLOCK AnalogInput
VAR_INPUT
    rawValue   : INT;         // Raw ADC value (0-1000)
    scaleLow   : INT;         // Engineering unit low
    scaleHigh  : INT;         // Engineering unit high
END_VAR
VAR_OUTPUT
    scaled     : INT;         // Scaled output in engineering units
    filtered   : INT;         // Filtered output (EMA)
    valid      : BOOL;        // TRUE if in valid range
END_VAR
VAR
    _filterState : INT := 0;
    _initialized : BOOL := FALSE;
END_VAR
    // Scale raw value to engineering units
    scaled := scaleLow + (rawValue * (scaleHigh - scaleLow)) / 1000;

    // Exponential moving average filter (alpha = 30%)
    IF NOT _initialized THEN
        _filterState := scaled;
        _initialized := TRUE;
    ELSE
        _filterState := (30 * scaled + 70 * _filterState) / 100;
    END_IF;
    filtered := _filterState;

    // Validity check
    IF rawValue >= 0 THEN
        IF rawValue <= 1000 THEN
            valid := TRUE;
        ELSE
            valid := FALSE;
        END_IF;
    ELSE
        valid := FALSE;
    END_IF;
END_FUNCTION_BLOCK

// ═══════════════════════════════════════════════════════════════════════
// FB: On/Off controller with hysteresis
// ═══════════════════════════════════════════════════════════════════════

FUNCTION_BLOCK HysteresisController
VAR_INPUT
    processValue : INT;
    setpoint     : INT;
    hysteresis   : INT;
END_VAR
VAR_OUTPUT
    output       : BOOL;
END_VAR
    IF processValue < (setpoint - hysteresis) THEN
        output := TRUE;    // Turn on
    ELSIF processValue > (setpoint + hysteresis) THEN
        output := FALSE;   // Turn off
    END_IF;
    // Otherwise maintain current state (hysteresis band)
END_FUNCTION_BLOCK

// ═══════════════════════════════════════════════════════════════════════
// FB: Configurable calculator with field-based I/O
// ═══════════════════════════════════════════════════════════════════════

FUNCTION_BLOCK Calculator
VAR_INPUT
    a   : INT;
    b   : INT;
    op  : INT;     // 0=add, 1=sub, 2=mul, 3=div
END_VAR
VAR_OUTPUT
    result : INT;
    error  : BOOL;
END_VAR
    error := FALSE;
    IF op = 0 THEN
        result := a + b;
    ELSIF op = 1 THEN
        result := a - b;
    ELSIF op = 2 THEN
        result := a * b;
    ELSIF op = 3 THEN
        IF b <> 0 THEN
            result := a / b;
        ELSE
            result := 0;
            error := TRUE;
        END_IF;
    ELSE
        result := 0;
        error := TRUE;
    END_IF;
END_FUNCTION_BLOCK

// ═══════════════════════════════════════════════════════════════════════
// Class: Alarm with trip count and configurable limits
// ═══════════════════════════════════════════════════════════════════════

CLASS Alarm
VAR
    _active     : BOOL := FALSE;
    _acked      : BOOL := FALSE;
    _tripCount  : INT := 0;
    _highLimit  : INT := 100;
    _hysteresis : INT := 5;
END_VAR

    PUBLIC METHOD Configure
    VAR_INPUT
        limit : INT;
        hyst  : INT;
    END_VAR
        _highLimit := limit;
        _hysteresis := hyst;
    END_METHOD

    PUBLIC METHOD Evaluate
    VAR_INPUT
        value : INT;
    END_VAR
    VAR
        wasActive : BOOL;
    END_VAR
        wasActive := _active;
        IF value > _highLimit THEN
            _active := TRUE;
        ELSIF value < (_highLimit - _hysteresis) THEN
            _active := FALSE;
        END_IF;
        // Count transitions to active
        IF _active AND NOT wasActive THEN
            _tripCount := _tripCount + 1;
            _acked := FALSE;
        END_IF;
    END_METHOD

    PUBLIC METHOD IsActive : INT
        IF _active THEN IsActive := 1; ELSE IsActive := 0; END_IF;
    END_METHOD

    PUBLIC METHOD GetTripCount : INT
        GetTripCount := _tripCount;
    END_METHOD

    PUBLIC METHOD Acknowledge
        _acked := TRUE;
    END_METHOD

    // Write alarm status through a pointer (out-param pattern)
    PUBLIC METHOD WriteStatus
    VAR_INPUT
        pActive : REF_TO INT;
        pTrips  : REF_TO INT;
    END_VAR
        IF pActive <> NULL THEN
            IF _active THEN pActive^ := 1; ELSE pActive^ := 0; END_IF;
        END_IF;
        IF pTrips <> NULL THEN
            pTrips^ := _tripCount;
        END_IF;
    END_METHOD
END_CLASS

// ═══════════════════════════════════════════════════════════════════════
// Class: Data logger with pointer-based sampling
// ═══════════════════════════════════════════════════════════════════════

CLASS DataLogger
VAR
    _sum   : INT := 0;
    _min   : INT := 32767;
    _max   : INT := -32768;
    _count : INT := 0;
END_VAR

    PUBLIC METHOD RecordFrom
    VAR_INPUT
        source : REF_TO INT;
    END_VAR
    VAR
        val : INT;
    END_VAR
        IF source <> NULL THEN
            val := source^;
            _sum := _sum + val;
            _count := _count + 1;
            IF val < _min THEN _min := val; END_IF;
            IF val > _max THEN _max := val; END_IF;
        END_IF;
    END_METHOD

    PUBLIC METHOD GetAverage : INT
        IF _count > 0 THEN
            GetAverage := _sum / _count;
        ELSE
            GetAverage := 0;
        END_IF;
    END_METHOD

    PUBLIC METHOD GetMin : INT
        GetMin := _min;
    END_METHOD

    PUBLIC METHOD GetMax : INT
        GetMax := _max;
    END_METHOD

    PUBLIC METHOD GetCount : INT
        GetCount := _count;
    END_METHOD

    PUBLIC METHOD Reset
        _sum := 0;
        _min := 32767;
        _max := -32768;
        _count := 0;
    END_METHOD
END_CLASS

// ═══════════════════════════════════════════════════════════════════════
// Main program: batch process with temperature control
// ═══════════════════════════════════════════════════════════════════════

VAR_GLOBAL
    // Analog input results
    g_raw_temp      : INT;
    g_scaled_temp   : INT;
    g_filtered_temp : INT;
    g_valid         : INT;

    // Controller
    g_heating       : INT;

    // Calculator
    g_calc_result   : INT;

    // Alarm
    g_alarm_active  : INT;
    g_alarm_trips   : INT;

    // Logger stats
    g_log_avg       : INT;
    g_log_min       : INT;
    g_log_max       : INT;
    g_log_count     : INT;

    // Cycle
    g_cycle         : INT;
END_VAR

PROGRAM Main
VAR
    // FB instances
    tempInput   : AnalogInput;
    controller  : HysteresisController;
    calc        : Calculator;

    // Class instances
    highTempAlarm : Alarm;
    tempLogger    : DataLogger;

    // Working variables
    cycle        : INT := 0;
    simRawAdc    : INT := 0;
    heaterOutput : INT := 0;
    alarmStatus  : INT := 0;
    alarmTrips   : INT := 0;
    dummy        : INT;
END_VAR
    cycle := cycle + 1;
    g_cycle := cycle;

    // ── Configure on first cycle ──
    IF cycle = 1 THEN
        highTempAlarm.Configure(limit := 80, hyst := 5);
    END_IF;

    // ── Simulate raw ADC reading ──
    // Ramp up, then stabilize, with some disturbance
    IF cycle < 20 THEN
        simRawAdc := cycle * 40;              // 0→800 over 20 cycles
    ELSE
        simRawAdc := 600;                     // Stabilize around 600
    END_IF;
    // Add cyclic disturbance
    IF (cycle MOD 4) < 2 THEN
        simRawAdc := simRawAdc + 50;
    ELSE
        simRawAdc := simRawAdc - 30;
    END_IF;
    // Apply heater effect (feedback)
    simRawAdc := simRawAdc + heaterOutput;
    dummy := ClampValue(target := REF(simRawAdc), lo := 0, hi := 1000);
    g_raw_temp := simRawAdc;

    // ── Process analog input (field-based I/O) ──
    tempInput.rawValue := simRawAdc;
    tempInput.scaleLow := 0;
    tempInput.scaleHigh := 100;
    tempInput();
    g_scaled_temp := tempInput.scaled;
    g_filtered_temp := tempInput.filtered;
    IF tempInput.valid THEN
        g_valid := 1;
    ELSE
        g_valid := 0;
    END_IF;

    // ── Hysteresis controller ──
    controller(processValue := tempInput.filtered,
               setpoint := 50,
               hysteresis := 5);
    IF controller.output THEN
        heaterOutput := 50;
        g_heating := 1;
    ELSE
        heaterOutput := 0;
        g_heating := 0;
    END_IF;

    // ── Calculator: compute temperature deviation ──
    calc.a := tempInput.filtered;
    calc.b := 50;
    calc.op := 1;     // subtract: deviation = filtered - setpoint
    calc();
    g_calc_result := calc.result;

    // ── Alarm evaluation ──
    highTempAlarm.Evaluate(value := tempInput.filtered);
    // Use pointer-based out-param pattern
    highTempAlarm.WriteStatus(pActive := REF(alarmStatus),
                              pTrips := REF(alarmTrips));
    g_alarm_active := alarmStatus;
    g_alarm_trips := alarmTrips;

    // ── Data logger: record filtered temperature ──
    // NOTE: REF(fb.field) is not yet supported — use intermediate variable
    alarmStatus := tempInput.filtered;
    tempLogger.RecordFrom(source := REF(alarmStatus));
    g_log_avg := tempLogger.GetAverage();
    g_log_min := tempLogger.GetMin();
    g_log_max := tempLogger.GetMax();
    g_log_count := tempLogger.GetCount();

    // Reset logger every 25 cycles
    IF (cycle MOD 25) = 0 THEN
        tempLogger.Reset();
    END_IF;
END_PROGRAM

(* ---- 14_class_instances.st ---- *)
(*
 * Class Instances — Lifecycle, Composition, and Interaction Patterns
 *
 * IEC 61131-3 classes are instantiated statically in VAR blocks (no NEW/heap).
 * This example demonstrates the full range of instance patterns:
 *
 * - Multiple independent instances of the same class
 * - Explicit initialization (constructor pattern)
 * - Init-once, run-many lifecycle
 * - Class instances inside function blocks (composition)
 * - Two classes interacting (producer-consumer)
 * - State machine lifecycle (idle → running → done → reset)
 * - Builder/configurator pattern
 * - Observer pattern: broadcast to multiple targets via pointers
 * - Inherited instances with independent state per level
 * - Reset and reuse across cycles
 *
 * Run with: st-cli run playground/14_class_instances.st -n 50
 *)

// ═══════════════════════════════════════════════════════════════════════
// Reusable class: Accumulator with reset
// ═══════════════════════════════════════════════════════════════════════

CLASS Accumulator
VAR
    _total : INT := 0;
    _count : INT := 0;
END_VAR

    PUBLIC METHOD Add
    VAR_INPUT v : INT; END_VAR
        _total := _total + v;
        _count := _count + 1;
    END_METHOD

    PUBLIC METHOD GetTotal : INT
        GetTotal := _total;
    END_METHOD

    PUBLIC METHOD GetCount : INT
        GetCount := _count;
    END_METHOD

    PUBLIC METHOD GetAverage : INT
        IF _count > 0 THEN
            GetAverage := _total / _count;
        ELSE
            GetAverage := 0;
        END_IF;
    END_METHOD

    PUBLIC METHOD Reset
        _total := 0;
        _count := 0;
    END_METHOD
END_CLASS

// ═══════════════════════════════════════════════════════════════════════
// State machine class — full lifecycle
// ═══════════════════════════════════════════════════════════════════════

CLASS BatchSequencer
VAR
    _state   : INT := 0;     // 0=idle, 1=filling, 2=heating, 3=mixing, 4=done
    _timer   : INT := 0;
    _target  : INT := 0;
    _product : INT := 0;     // accumulated product
END_VAR

    PUBLIC METHOD Start
    VAR_INPUT batchSize : INT; END_VAR
        IF _state = 0 THEN
            _state := 1;
            _timer := 0;
            _target := batchSize;
            _product := 0;
        END_IF;
    END_METHOD

    PUBLIC METHOD Update
        IF _state = 1 THEN
            // Filling
            _product := _product + 10;
            _timer := _timer + 1;
            IF _product >= _target THEN
                _state := 2;
                _timer := 0;
            END_IF;
        ELSIF _state = 2 THEN
            // Heating
            _timer := _timer + 1;
            IF _timer >= 5 THEN
                _state := 3;
                _timer := 0;
            END_IF;
        ELSIF _state = 3 THEN
            // Mixing
            _timer := _timer + 1;
            IF _timer >= 3 THEN
                _state := 4;
            END_IF;
        END_IF;
    END_METHOD

    PUBLIC METHOD GetState : INT
        GetState := _state;
    END_METHOD

    PUBLIC METHOD GetProduct : INT
        GetProduct := _product;
    END_METHOD

    PUBLIC METHOD IsDone : INT
        IF _state = 4 THEN IsDone := 1; ELSE IsDone := 0; END_IF;
    END_METHOD

    PUBLIC METHOD Reset
        _state := 0;
        _timer := 0;
        _product := 0;
    END_METHOD
END_CLASS

// ═══════════════════════════════════════════════════════════════════════
// Producer-Consumer pattern
// ═══════════════════════════════════════════════════════════════════════

CLASS Producer
VAR
    _sequence : INT := 0;
END_VAR
    PUBLIC METHOD Produce : INT
        _sequence := _sequence + 7;
        Produce := _sequence;
    END_METHOD
    PUBLIC METHOD GetSequence : INT
        GetSequence := _sequence;
    END_METHOD
END_CLASS

CLASS Consumer
VAR
    _consumed : INT := 0;
    _items    : INT := 0;
END_VAR
    PUBLIC METHOD Consume
    VAR_INPUT amount : INT; END_VAR
        _consumed := _consumed + amount;
        _items := _items + 1;
    END_METHOD
    PUBLIC METHOD GetConsumed : INT
        GetConsumed := _consumed;
    END_METHOD
    PUBLIC METHOD GetItems : INT
        GetItems := _items;
    END_METHOD
END_CLASS

// ═══════════════════════════════════════════════════════════════════════
// Observer pattern — broadcast values via pointers
// ═══════════════════════════════════════════════════════════════════════

CLASS Broadcaster
VAR
    _value : INT := 0;
END_VAR
    PUBLIC METHOD SetValue
    VAR_INPUT v : INT; END_VAR
        _value := v;
    END_METHOD
    PUBLIC METHOD Notify
    VAR_INPUT
        p1 : REF_TO INT;
        p2 : REF_TO INT;
        p3 : REF_TO INT;
    END_VAR
        IF p1 <> NULL THEN p1^ := _value; END_IF;
        IF p2 <> NULL THEN p2^ := _value; END_IF;
        IF p3 <> NULL THEN p3^ := _value; END_IF;
    END_METHOD
END_CLASS

// ═══════════════════════════════════════════════════════════════════════
// FB wrapper with class inside (composition)
// ═══════════════════════════════════════════════════════════════════════

FUNCTION_BLOCK SensorChannel
VAR_INPUT
    rawValue : INT;
END_VAR
VAR_OUTPUT
    filtered : INT;
    sampleCount : INT;
END_VAR
VAR
    stats : Accumulator;
END_VAR
    stats.Add(v := rawValue);
    filtered := stats.GetAverage();
    sampleCount := stats.GetCount();
END_FUNCTION_BLOCK

// ═══════════════════════════════════════════════════════════════════════
// Inheritance: base controller → specialized controller
// ═══════════════════════════════════════════════════════════════════════

CLASS BaseController
VAR
    _output : INT := 0;
    _enabled : BOOL := FALSE;
END_VAR
    PUBLIC METHOD Enable
        _enabled := TRUE;
    END_METHOD
    PUBLIC METHOD Disable
        _enabled := FALSE;
        _output := 0;
    END_METHOD
    PUBLIC METHOD GetOutput : INT
        GetOutput := _output;
    END_METHOD
    PUBLIC METHOD IsEnabled : INT
        IF _enabled THEN IsEnabled := 1; ELSE IsEnabled := 0; END_IF;
    END_METHOD
END_CLASS

CLASS BangBangController EXTENDS BaseController
VAR
    _setpoint : INT := 50;
    _hysteresis : INT := 5;
END_VAR
    PUBLIC METHOD Configure
    VAR_INPUT sp : INT; hyst : INT; END_VAR
        _setpoint := sp;
        _hysteresis := hyst;
    END_METHOD
    PUBLIC METHOD Compute
    VAR_INPUT pv : INT; END_VAR
        IF _enabled THEN
            IF pv < (_setpoint - _hysteresis) THEN
                _output := 100;
            ELSIF pv > (_setpoint + _hysteresis) THEN
                _output := 0;
            END_IF;
        ELSE
            _output := 0;
        END_IF;
    END_METHOD
END_CLASS

// ═══════════════════════════════════════════════════════════════════════
// Main program
// ═══════════════════════════════════════════════════════════════════════

VAR_GLOBAL
    // Multiple accumulators
    g_fast_total   : INT;
    g_slow_total   : INT;

    // Batch sequencer
    g_batch_state  : INT;
    g_batch_done   : INT;
    g_batch_product : INT;

    // Producer-Consumer
    g_produced     : INT;
    g_consumed     : INT;

    // Observer
    g_obs_a        : INT;
    g_obs_b        : INT;
    g_obs_c        : INT;

    // Sensor channel (FB with class)
    g_ch1_avg      : INT;
    g_ch2_avg      : INT;
    g_ch1_samples  : INT;
    g_ch2_samples  : INT;

    // Controller
    g_ctrl_out     : INT;

    g_cycle        : INT;
END_VAR

PROGRAM Main
VAR
    // Multiple independent instances
    fastAcc   : Accumulator;
    slowAcc   : Accumulator;

    // State machine
    batch     : BatchSequencer;

    // Producer-Consumer
    producer  : Producer;
    consumer  : Consumer;
    item      : INT;

    // Observer
    broadcast : Broadcaster;
    obs_a : INT := 0;
    obs_b : INT := 0;
    obs_c : INT := 0;

    // FB with class inside — two independent channels
    ch1 : SensorChannel;
    ch2 : SensorChannel;

    // Inherited controller
    ctrl : BangBangController;

    cycle : INT := 0;
    simTemp : INT := 30;
END_VAR
    cycle := cycle + 1;
    g_cycle := cycle;

    // ── Multiple independent accumulators ──
    fastAcc.Add(v := 10);
    IF (cycle MOD 3) = 0 THEN
        slowAcc.Add(v := 100);
    END_IF;
    g_fast_total := fastAcc.GetTotal();
    g_slow_total := slowAcc.GetTotal();
    // Reset fast accumulator every 10 cycles
    IF (cycle MOD 10) = 0 THEN
        fastAcc.Reset();
    END_IF;

    // ── Batch sequencer lifecycle ──
    IF cycle = 1 THEN
        batch.Start(batchSize := 50);
    END_IF;
    batch.Update();
    g_batch_state := batch.GetState();
    g_batch_done := batch.IsDone();
    g_batch_product := batch.GetProduct();
    // Restart if done
    IF batch.IsDone() = 1 THEN
        batch.Reset();
        batch.Start(batchSize := 50);
    END_IF;

    // ── Producer-Consumer ──
    item := producer.Produce();
    consumer.Consume(amount := item);
    g_produced := item;
    g_consumed := consumer.GetConsumed();

    // ── Observer broadcast ──
    broadcast.SetValue(v := cycle * 11);
    broadcast.Notify(p1 := REF(obs_a), p2 := REF(obs_b), p3 := REF(obs_c));
    g_obs_a := obs_a;
    g_obs_b := obs_b;
    g_obs_c := obs_c;

    // ── Two sensor channels with class inside FB ──
    ch1(rawValue := 100 + cycle);
    ch2(rawValue := 200 + cycle * 2);
    g_ch1_avg := ch1.filtered;
    g_ch2_avg := ch2.filtered;
    g_ch1_samples := ch1.sampleCount;
    g_ch2_samples := ch2.sampleCount;

    // ── Inherited controller ──
    IF cycle = 1 THEN
        ctrl.Configure(sp := 50, hyst := 5);
        ctrl.Enable();
    END_IF;
    // Simulate temperature responding to controller
    IF g_ctrl_out > 50 THEN
        simTemp := simTemp + 2;
    ELSIF simTemp > 30 THEN
        simTemp := simTemp - 1;
    END_IF;
    ctrl.Compute(pv := simTemp);
    g_ctrl_out := ctrl.GetOutput();
END_PROGRAM

(* ---- 01_hello.st ---- *)
(*
 * Hello World — Minimal ST program
 * Open this file to test diagnostics, hover, and go-to-definition.
 *)

PROGRAM HelloWorld
VAR
    counter : INT := 0;
    realCounter : REAL := 0;
    rad : REAL;
    running : BOOL := TRUE;
    seno : LREAL := 0;
END_VAR

    IF running THEN
        counter := counter + 1;
        realCounter := counter;
        rad := (realCounter/180.0) * 3.1415;
        seno := SIN(rad);
        IF counter > 1000 THEN
            running := FALSE;
        END_IF;
    END_IF;
END_PROGRAM

(* ---- 05_errors_demo.st ---- *)
(*
 * Error showcase — intentionally broken code to demonstrate diagnostics.
 * Open this file to see the LSP reporting errors and warnings in real time.
 *
 * Try fixing the errors one by one and watch diagnostics update!
 *)

PROGRAM ErrorShowcase
VAR
    x : INT := 0;
    b : BOOL := TRUE;
    unused_var : REAL := 3.14;  // ⚠ unused variable warning
END_VAR
    // ❌ Error: undeclared variable
    x := undeclared_variable;

    // ❌ Error: type mismatch — assigning BOOL to INT
    x := b;

    // ❌ Error: condition must be BOOL, not INT
    IF x THEN
        x := 0;
    END_IF;

    // ❌ Error: EXIT outside of a loop
    EXIT;

    // ❌ Error: calling something that isn't a function
    x := x(a := 1);
END_PROGRAM

(* ---- 07_stdlib_demo.st ---- *)
(*
 * Standard Library Demo
 *
 * Demonstrates the built-in standard library modules:
 * - CTU (count up), CTD (count down), CTUD (count up/down)
 * - R_TRIG (rising edge), F_TRIG (falling edge)
 * - TON (on-delay timer), TOF (off-delay timer), TP (pulse timer)
 * - Math: MAX_INT, MIN_INT, LIMIT_INT, ABS_INT, SEL
 * - Conversion: BOOL_TO_INT, INT_TO_BOOL
 *
 * Run with: st-cli run playground/07_stdlib_demo.st -n 50
 *)

VAR_GLOBAL
    g_bottle_count : INT;
    g_timer_done : INT;
    g_edge_count : INT;
END_VAR

PROGRAM StdlibDemo
VAR
    // ── Counters ──
    bottle_counter : CTU;       // Counts bottles on conveyor
    reject_counter : CTD;       // Counts down rejects remaining

    // ── Edge detection ──
    sensor_edge : R_TRIG;       // Detects new bottle arrival
    clear_edge : F_TRIG;        // Detects sensor clear

    // ── Timers ──
    fill_timer : TON;           // Delay before fill starts
    hold_timer : TP;            // Pulse output for gripper

    // ── Process variables ──
    cycle : INT := 0;
    sensor : BOOL := FALSE;
    filling : BOOL := FALSE;
    clamped_speed : INT := 0;
    edge_events : INT := 0;
END_VAR
    cycle := cycle + 1;

    // Simulate sensor: bottle arrives every 10 cycles, stays for 3 cycles
    sensor := (cycle MOD 10) >= 0 AND (cycle MOD 10) < 3;

    // ── Edge detection: count sensor transitions ──
    sensor_edge(CLK := sensor);
    clear_edge(CLK := sensor);
    IF sensor_edge.Q THEN
        edge_events := edge_events + 1;
    END_IF;

    // ── Counter: count bottles ──
    bottle_counter(CU := sensor_edge.Q, RESET := FALSE, PV := 100);

    // ── Timer: delay filling by 5 cycles after sensor ──
    fill_timer(IN1 := sensor, PT := 5);
    filling := fill_timer.Q;

    // ── Pulse: gripper activates for 3 cycles on each bottle ──
    hold_timer(IN1 := sensor_edge.Q, PT := 3);

    // ── Math: clamp conveyor speed ──
    clamped_speed := LIMIT_INT(MN := 10, IN1 := cycle, MX := 100);

    // ── Selection: choose mode based on counter ──
    g_bottle_count := bottle_counter.CV;
    g_timer_done := BOOL_TO_INT(IN1 := filling);
    g_edge_count := edge_events;
END_PROGRAM

(* ---- 09_pointers.st ---- *)
(*
 * Pointers and References — REF_TO and ^ dereference operator
 *
 * Demonstrates IEC 61131-3 pointer support:
 * - REF_TO <type>  declares a typed pointer variable
 * - REF(variable)  takes the reference (address) of a variable
 * - ptr^           dereferences a pointer (read or write)
 * - NULL           null pointer literal
 *
 * Run with: st-cli run playground/09_pointers.st -n 10
 *)

VAR_GLOBAL
    g_direct_value : INT;
    g_via_pointer : INT;
    g_swapped_a : INT;
    g_swapped_b : INT;
END_VAR

// ── Swap two integers using pointers ─────────────────────────────────
// This demonstrates how pointers enable generic operations
// on variables without knowing their names at compile time.

FUNCTION SwapInt : INT
VAR_INPUT
    p1 : REF_TO INT;
    p2 : REF_TO INT;
END_VAR
VAR
    temp : INT := 0;
END_VAR
    temp := p1^;
    p1^ := p2^;
    p2^ := temp;
    SwapInt := 0;
END_FUNCTION

// ── Indirect write: modify a variable through a pointer ──────────────

FUNCTION IncrementVia : INT
VAR_INPUT
    target : REF_TO INT;
    amount : INT;
END_VAR
    IF target <> NULL THEN
        target^ := target^ + amount;
    END_IF;
    IncrementVia := target^;
END_FUNCTION

// ── Main Program ─────────────────────────────────────────────────────

PROGRAM Main
VAR
    counter : INT := 0;
    value_a : INT := 100;
    value_b : INT := 200;

    ptr : REF_TO INT;
    null_ptr : REF_TO INT;

    cycle : INT := 0;
    dummy : INT := 0;
END_VAR
    cycle := cycle + 1;

    // ── Basic pointer usage ──
    // Take a reference and read through it
    ptr := REF(counter);
    counter := counter + 1;
    g_direct_value := counter;
    g_via_pointer := ptr^;         // Same value, accessed via pointer

    // ── Indirect modification ──
    // Modify counter through the pointer
    dummy := IncrementVia(target := REF(counter), amount := 10);

    // ── Swap two values using pointers ──
    // Every 5 cycles, swap value_a and value_b
    IF (cycle MOD 5) = 0 THEN
        dummy := SwapInt(p1 := REF(value_a), p2 := REF(value_b));
    END_IF;

    g_swapped_a := value_a;
    g_swapped_b := value_b;

    // ── NULL safety ──
    // Dereferencing NULL returns 0 (safe, no crash)
    null_ptr := NULL;
    dummy := null_ptr^;            // Returns 0
END_PROGRAM

(* ---- 15_mandelbrot.st ---- *)
(*
 * Mandelbrot set — ASCII art rendered one row per scan cycle.
 *
 * Computes the classic Mandelbrot fractal over the region
 * [-2.0, 0.8] x [-1.2, 1.2] on an 80x40 character grid.
 * Each scan cycle computes one full row (80 pixels).
 * After 40 cycles the entire image is done and it restarts.
 *
 * The escape-time algorithm iterates z = z^2 + c for each pixel,
 * counting how many iterations before |z| > 2.0 (max 80).
 * The iteration count maps to an ASCII density character.
 *
 * Run:
 *   st-cli run playground/15_mandelbrot.st -n 42
 *)

VAR_GLOBAL
    (* Current row being rendered (0..39) *)
    g_row        : INT := 0;
    (* Total rows completed *)
    g_rows_done  : INT := 0;
    (* Pixels computed this cycle *)
    g_pixels     : INT := 0;
    (* Total escape iterations across all pixels (measures "complexity") *)
    g_total_iters : INT := 0;
    (* Max iterations hit by any single pixel *)
    g_max_iters   : INT := 0;
    (* Count of pixels inside the set (didn't escape) *)
    g_inside_count : INT := 0;
END_VAR

(*
 * Mandelbrot escape-time computation for a single point.
 * Returns the number of iterations before |z| > 2.0,
 * or max_iter if the point is inside the set.
 *)
FUNCTION MandelbrotEscape : INT
VAR_INPUT
    cx       : REAL;    (* Real part of c *)
    cy       : REAL;    (* Imaginary part of c *)
    max_iter : INT;     (* Maximum iterations *)
END_VAR
VAR
    zr   : REAL := 0.0;   (* Real part of z *)
    zi   : REAL := 0.0;   (* Imaginary part of z *)
    zr2  : REAL;           (* zr * zr — cached to avoid recomputation *)
    zi2  : REAL;           (* zi * zi *)
    iter : INT  := 0;
END_VAR
    (* z = 0 + 0i, iterate z := z^2 + c *)
    WHILE iter < max_iter DO
        zr2 := zr * zr;
        zi2 := zi * zi;

        (* Escape condition: |z|^2 > 4.0 *)
        IF (zr2 + zi2) > 4.0 THEN
            MandelbrotEscape := iter;
            RETURN;
        END_IF;

        (* z := z^2 + c
           (a + bi)^2 = a^2 - b^2 + 2abi *)
        zi := 2.0 * zr * zi + cy;
        zr := zr2 - zi2 + cx;

        iter := iter + 1;
    END_WHILE;

    (* Point is inside the set *)
    MandelbrotEscape := max_iter;
END_FUNCTION

(*
 * Map an iteration count to an ASCII density character index.
 * 0 = space (inside set), higher = denser glyph.
 * We return an INT index into a conceptual palette:
 *   0: ' '  (inside the Mandelbrot set)
 *   1: '.'  2: ':'  3: '-'  4: '='  5: '+'
 *   6: '*'  7: '#'  8: '%'  9: '@'
 *)
FUNCTION IterToGlyph : INT
VAR_INPUT
    iters    : INT;
    max_iter : INT;
END_VAR
    IF iters >= max_iter THEN
        IterToGlyph := 0;    (* Inside set *)
    ELSIF iters < 2 THEN
        IterToGlyph := 9;    (* Very fast escape = dense *)
    ELSIF iters < 4 THEN
        IterToGlyph := 8;
    ELSIF iters < 8 THEN
        IterToGlyph := 7;
    ELSIF iters < 12 THEN
        IterToGlyph := 6;
    ELSIF iters < 20 THEN
        IterToGlyph := 5;
    ELSIF iters < 30 THEN
        IterToGlyph := 4;
    ELSIF iters < 45 THEN
        IterToGlyph := 3;
    ELSIF iters < 60 THEN
        IterToGlyph := 2;
    ELSE
        IterToGlyph := 1;
    END_IF;
END_FUNCTION

(*
 * Main program — computes one row of the Mandelbrot set per scan cycle.
 *
 * Grid: 80 columns x 40 rows
 * Region: x in [-2.0, 0.8], y in [-1.2, 1.2]
 *)
PROGRAM Main
VAR
    col       : INT;
    cx        : REAL;
    cy        : REAL;
    iters     : INT;
    glyph     : INT;
    row_max   : INT := 0;
    row_inside : INT := 0;
    row_iters  : INT := 0;
END_VAR
    (* Map current row to imaginary axis: y in [-1.2, 1.2] *)
    cy := 1.2 - (INT_TO_REAL(IN1 := g_row) * 2.4 / 40.0);

    row_max := 0;
    row_inside := 0;
    row_iters := 0;
    g_pixels := 0;

    FOR col := 0 TO 79 DO
        (* Map column to real axis: x in [-2.0, 0.8] *)
        cx := -2.0 + (INT_TO_REAL(IN1 := col) * 2.8 / 80.0);

        (* Compute escape time *)
        iters := MandelbrotEscape(cx := cx, cy := cy, max_iter := 80);

        (* Track stats *)
        row_iters := row_iters + iters;
        IF iters > row_max THEN
            row_max := iters;
        END_IF;
        IF iters >= 80 THEN
            row_inside := row_inside + 1;
        END_IF;

        (* Convert to ASCII glyph index *)
        glyph := IterToGlyph(iters := iters, max_iter := 80);

        g_pixels := g_pixels + 1;
    END_FOR;

    (* Update globals *)
    g_total_iters := g_total_iters + row_iters;
    g_inside_count := g_inside_count + row_inside;
    IF row_max > g_max_iters THEN
        g_max_iters := row_max;
    END_IF;

    g_rows_done := g_rows_done + 1;
    g_row := g_row + 1;

    (* Wrap around after 40 rows — restart the render *)
    IF g_row >= 40 THEN
        g_row := 0;
    END_IF;
END_PROGRAM

(* ---- 16_time_conversions.st ---- *)
(*
 * Playground 16: Time & Type Conversion Functions
 *
 * Demonstrates all TIME_TO_*, *_TO_TIME, and generic TO_*/ANY_TO_*
 * conversion functions. TIME values are stored as milliseconds (i64).
 *
 * Run with: st-cli run playground/16_time_conversions.st
 *)

VAR_GLOBAL
    (* TIME_TO_* results *)
    g_time_to_int    : INT;
    g_time_to_dint   : INT;
    g_time_to_lint   : INT;
    g_time_to_sint   : INT;    (* SINT narrowing at VM level *)
    g_time_to_real   : REAL;
    g_time_to_lreal  : LREAL;
    g_time_to_bool_t : INT;   (* BOOL as INT for output *)
    g_time_to_bool_f : INT;

    (* *_TO_TIME results — stored as INT for easy verification *)
    g_int_to_time    : INT;
    g_dint_to_time   : INT;
    g_lint_to_time   : INT;
    g_real_to_time   : INT;
    g_bool_to_time_t : INT;
    g_bool_to_time_f : INT;

    (* Overloaded TO_* results *)
    g_to_int_from_time  : INT;
    g_to_real_from_time : REAL;
    g_to_bool_from_time : INT;
    g_to_time_from_int  : INT;

    (* ANY_TO_* results *)
    g_any_to_int_from_time  : INT;
    g_any_to_real_from_time : REAL;
    g_any_to_bool_from_time : INT;
    g_any_to_time_from_int  : INT;

    (* Round-trip verification *)
    g_roundtrip_int  : INT;    (* TIME -> INT -> TIME -> INT *)
    g_roundtrip_real : INT;    (* TIME -> REAL -> TIME -> INT *)

    (* Arithmetic with converted values *)
    g_time_sum : INT;
    g_time_diff : INT;

    (* Edge cases *)
    g_zero_time  : INT;
    g_large_time : DINT;
END_VAR

PROGRAM Main
VAR
    t5s       : TIME := T#5s;          (* 5000 ms *)
    t100ms    : TIME := T#100ms;       (* 100 ms *)
    t0        : TIME := T#0ms;         (* 0 ms *)
    t1d2h     : TIME := T#1d2h3m4s5ms; (* 93784005 ms *)
    ms_val    : INT;
    t_from_ms : TIME;
    t_sum     : TIME;
END_VAR
    (* ── TIME_TO_* ─────────────────────────────────────────────── *)
    g_time_to_int   := TIME_TO_INT(IN1 := t5s);         (* 5000 *)
    g_time_to_dint  := TIME_TO_DINT(IN1 := t5s);        (* 5000 *)
    g_time_to_lint  := TIME_TO_LINT(IN1 := t5s);        (* 5000 *)
    g_time_to_sint  := TIME_TO_SINT(IN1 := t100ms);     (* 100 *)
    g_time_to_real  := TIME_TO_REAL(IN1 := t5s);        (* 5000.0 *)
    g_time_to_lreal := TIME_TO_LREAL(IN1 := t5s);       (* 5000.0 *)
    g_time_to_bool_t := BOOL_TO_INT(IN1 := TIME_TO_BOOL(IN1 := t5s));   (* TRUE -> 1 *)
    g_time_to_bool_f := BOOL_TO_INT(IN1 := TIME_TO_BOOL(IN1 := t0));    (* FALSE -> 0 *)

    (* ── *_TO_TIME ─────────────────────────────────────────────── *)
    g_int_to_time    := TIME_TO_INT(IN1 := INT_TO_TIME(IN1 := 3000));    (* 3000 *)
    g_dint_to_time   := TIME_TO_INT(IN1 := DINT_TO_TIME(IN1 := 7500));   (* 7500 *)
    g_lint_to_time   := TIME_TO_INT(IN1 := LINT_TO_TIME(IN1 := 12000));  (* 12000 *)
    g_real_to_time   := TIME_TO_INT(IN1 := REAL_TO_TIME(IN1 := 2500.0)); (* 2500 *)
    g_bool_to_time_t := TIME_TO_INT(IN1 := BOOL_TO_TIME(IN1 := TRUE));   (* 1 *)
    g_bool_to_time_f := TIME_TO_INT(IN1 := BOOL_TO_TIME(IN1 := FALSE));  (* 0 *)

    (* ── Overloaded TO_* ───────────────────────────────────────── *)
    g_to_int_from_time  := TO_INT(IN1 := t100ms);           (* 100 *)
    g_to_real_from_time := TO_REAL(IN1 := t5s);              (* 5000.0 *)
    g_to_bool_from_time := BOOL_TO_INT(IN1 := TO_BOOL(IN1 := t5s));  (* 1 *)
    g_to_time_from_int  := TIME_TO_INT(IN1 := TO_TIME(IN1 := 4000)); (* 4000 *)

    (* ── ANY_TO_* ──────────────────────────────────────────────── *)
    g_any_to_int_from_time  := ANY_TO_INT(IN1 := t100ms);           (* 100 *)
    g_any_to_real_from_time := ANY_TO_REAL(IN1 := t5s);              (* 5000.0 *)
    g_any_to_bool_from_time := BOOL_TO_INT(IN1 := ANY_TO_BOOL(IN1 := t5s));  (* 1 *)
    g_any_to_time_from_int  := TIME_TO_INT(IN1 := ANY_TO_TIME(IN1 := 6000)); (* 6000 *)

    (* ── Round-trip verification ───────────────────────────────── *)
    (* TIME -> INT -> TIME -> INT should preserve value *)
    ms_val    := TIME_TO_INT(IN1 := t5s);                   (* 5000 *)
    t_from_ms := INT_TO_TIME(IN1 := ms_val);                (* T#5s *)
    g_roundtrip_int := TIME_TO_INT(IN1 := t_from_ms);       (* 5000 *)

    (* TIME -> REAL -> TIME -> INT should be close (float precision) *)
    g_roundtrip_real := TIME_TO_INT(IN1 := REAL_TO_TIME(IN1 := TIME_TO_REAL(IN1 := t5s))); (* 5000 *)

    (* ── Arithmetic with converted values ──────────────────────── *)
    t_sum := t5s + t100ms;
    g_time_sum := TIME_TO_INT(IN1 := t_sum);                (* 5100 *)
    g_time_diff := TIME_TO_INT(IN1 := t5s - t100ms);        (* 4900 *)

    (* ── Edge cases ────────────────────────────────────────────── *)
    g_zero_time := TIME_TO_INT(IN1 := t0);                   (* 0 *)
    g_large_time := TIME_TO_DINT(IN1 := t1d2h);              (* 93784005 *)
END_PROGRAM

(* ---- 17_date_time_types.st ---- *)
(*
 * Playground 17: DATE, TOD, DT Types & Conversions
 *
 * Demonstrates DATE/TOD/DT literal parsing, conversions to/from
 * numeric types, cross-type extraction (DT_TO_DATE, DT_TO_TOD),
 * date/time arithmetic, CONCAT_DATE_TOD, MULTIME, DIVTIME,
 * DAY_OF_WEEK, and TO_*/ANY_TO_* generic conversions.
 *
 * All date/time types are stored internally as milliseconds (i64).
 * DATE = ms since epoch, TOD = ms since midnight, DT = ms since epoch.
 * Use LINT for date/DT values as ms since epoch exceeds DINT range.
 *)

VAR_GLOBAL
    (* DATE literal parsing — LINT needed, values exceed DINT range *)
    g_date_ms       : LINT;   (* D#2024-01-15 → ms since epoch *)
    g_date_epoch    : LINT;   (* D#1970-01-01 → 0 *)

    (* TOD literal parsing — DINT is sufficient (max ~86M ms) *)
    g_tod_ms        : DINT;   (* TOD#12:30:00 → 45000000 ms *)
    g_tod_midnight  : DINT;   (* TOD#00:00:00 → 0 *)
    g_tod_frac      : DINT;   (* TOD#12:30:00.500 → 45000500 ms *)

    (* DT literal parsing *)
    g_dt_ms         : LINT;   (* DT#2024-01-15-12:30:00 *)

    (* DATE_TO_* *)
    g_date_to_int   : LINT;
    g_date_to_real  : REAL;
    g_date_to_bool  : INT;

    (* TOD_TO_* *)
    g_tod_to_int    : DINT;
    g_tod_to_real   : REAL;

    (* DT extraction *)
    g_dt_to_date    : LINT;   (* date portion *)
    g_dt_to_tod     : DINT;   (* tod portion *)

    (* CONCAT_DATE_TOD *)
    g_concat_dt     : LINT;

    (* Date/time arithmetic *)
    g_add_tod_time  : DINT;   (* TOD + TIME *)
    g_sub_tod_time  : DINT;   (* TOD - TIME *)
    g_sub_date_date : LINT;   (* DATE - DATE → TIME ms *)
    g_sub_dt_dt     : DINT;   (* DT - DT → TIME ms, small diff *)
    g_add_dt_time   : LINT;   (* DT + TIME *)

    (* MULTIME / DIVTIME *)
    g_multime       : DINT;
    g_divtime       : DINT;

    (* DAY_OF_WEEK *)
    g_dow_thu       : INT;    (* 1970-01-01 = Thursday = 4 *)
    g_dow_sun       : INT;    (* 1970-01-04 = Sunday = 0 *)
    g_dow_mon       : INT;    (* 2024-01-15 = Monday = 1 *)

    (* Generic TO_*/ANY_TO_* *)
    g_to_date       : LINT;
    g_any_to_tod    : DINT;
    g_any_to_dt     : LINT;

    (* Round-trip: DT → DATE + TOD → CONCAT → DT *)
    g_roundtrip_dt  : LINT;
END_VAR

PROGRAM Main
VAR
    d1    : DATE := D#2024-01-15;
    d2    : DATE := D#1970-01-01;
    d3    : DATE := D#1970-01-04;  (* Sunday *)
    t1    : TOD  := TOD#12:30:00;
    t2    : TOD  := TOD#00:00:00;
    t3    : TOD  := TOD#12:30:00.500;
    dt1   : DT   := DT#2024-01-15-12:30:00;
    dur   : TIME := T#1h;
    d_part : DATE;
    t_part : TOD;
END_VAR
    (* ── Literal parsing verification ──────────────────────────── *)
    g_date_ms     := DATE_TO_LINT(IN1 := d1);
    g_date_epoch  := DATE_TO_LINT(IN1 := d2);
    g_tod_ms      := TOD_TO_DINT(IN1 := t1);
    g_tod_midnight := TOD_TO_DINT(IN1 := t2);
    g_tod_frac    := TOD_TO_DINT(IN1 := t3);
    g_dt_ms       := DT_TO_LINT(IN1 := dt1);

    (* ── DATE_TO_* / TOD_TO_* ─────────────────────────────────── *)
    g_date_to_int  := DATE_TO_LINT(IN1 := d1);
    g_date_to_real := DATE_TO_REAL(IN1 := d1);
    g_date_to_bool := BOOL_TO_INT(IN1 := DATE_TO_BOOL(IN1 := d1));
    g_tod_to_int   := TOD_TO_DINT(IN1 := t1);
    g_tod_to_real  := TOD_TO_REAL(IN1 := t1);

    (* ── DT extraction ────────────────────────────────────────── *)
    g_dt_to_date := DATE_TO_LINT(IN1 := DT_TO_DATE(IN1 := dt1));
    g_dt_to_tod  := TOD_TO_DINT(IN1 := DT_TO_TOD(IN1 := dt1));

    (* ── CONCAT_DATE_TOD ──────────────────────────────────────── *)
    g_concat_dt := DT_TO_LINT(IN1 := CONCAT_DATE_TOD(IN1 := d1, IN2 := t1));

    (* ── Date/time arithmetic ─────────────────────────────────── *)
    g_add_tod_time  := TOD_TO_DINT(IN1 := ADD_TOD_TIME(IN1 := t1, IN2 := dur));
    g_sub_tod_time  := TOD_TO_DINT(IN1 := SUB_TOD_TIME(IN1 := t1, IN2 := dur));
    g_sub_date_date := TIME_TO_LINT(IN1 := SUB_DATE_DATE(IN1 := d1, IN2 := d2));
    g_sub_dt_dt     := TIME_TO_DINT(IN1 := SUB_DT_DT(IN1 := dt1, IN2 :=
                            CONCAT_DATE_TOD(IN1 := d1, IN2 := t2)));
    g_add_dt_time   := DT_TO_LINT(IN1 := ADD_DT_TIME(IN1 := dt1, IN2 := dur));

    (* ── MULTIME / DIVTIME ────────────────────────────────────── *)
    g_multime := TIME_TO_DINT(IN1 := MULTIME(IN1 := T#1s, IN2 := 5));
    g_divtime := TIME_TO_DINT(IN1 := DIVTIME(IN1 := T#10s, IN2 := 2));

    (* ── DAY_OF_WEEK ──────────────────────────────────────────── *)
    g_dow_thu := DAY_OF_WEEK(IN1 := d2);        (* 1970-01-01 = Thursday = 4 *)
    g_dow_sun := DAY_OF_WEEK(IN1 := d3);        (* 1970-01-04 = Sunday = 0 *)
    g_dow_mon := DAY_OF_WEEK(IN1 := d1);        (* 2024-01-15 = Monday = 1 *)

    (* ── Generic TO_*/ANY_TO_* ────────────────────────────────── *)
    g_to_date   := DATE_TO_LINT(IN1 := TO_DATE(IN1 := 0));
    g_any_to_tod := TOD_TO_DINT(IN1 := ANY_TO_TOD(IN1 := 45000000));
    g_any_to_dt  := DT_TO_LINT(IN1 := ANY_TO_DT(IN1 := 1000));

    (* ── Round-trip: DT → split → concat → verify ─────────────── *)
    d_part := DT_TO_DATE(IN1 := dt1);
    t_part := DT_TO_TOD(IN1 := dt1);
    g_roundtrip_dt := DT_TO_LINT(IN1 := CONCAT_DATE_TOD(IN1 := d_part, IN2 := t_part));
END_PROGRAM

(* ---- 18_strings.st ---- *)
(*
 * Playground 18: String Manipulation & Formatting
 *
 * Demonstrates every IEC 61131-3 / CODESYS-compatible string function:
 *   - Core: LEN, LEFT, RIGHT, MID, CONCAT, INSERT, DELETE, REPLACE, FIND
 *   - Case: TO_UPPER, TO_LOWER (and aliases UPPER_CASE, LOWER_CASE)
 *   - Trim: TRIM, LTRIM, RTRIM
 *   - Numeric ↔ STRING: *_TO_STRING, STRING_TO_*, generic TO_STRING
 *
 * Each global below has a deterministic expected value; the matching
 * E2E test in stdlib_tests.rs (`playground_18_strings_e2e`) asserts
 * every one of them.
 *
 * Run with: st-cli run playground/18_strings.st
 *)

VAR_GLOBAL
    (* LEN *)
    g_len_hello   : INT;
    g_len_empty   : INT;

    (* LEFT / RIGHT — including out-of-range clamping *)
    g_left_3      : STRING;
    g_left_zero   : STRING;
    g_left_huge   : STRING;
    g_left_neg    : STRING;
    g_right_3     : STRING;
    g_right_zero  : STRING;
    g_right_huge  : STRING;

    (* MID — including edge cases *)
    g_mid_mid     : STRING;
    g_mid_start   : STRING;
    g_mid_end     : STRING;
    g_mid_overrun : STRING;
    g_mid_pos0    : STRING;
    g_mid_negpos  : STRING;
    g_mid_zerolen : STRING;

    (* CONCAT *)
    g_concat      : STRING;
    g_concat_empty: STRING;

    (* INSERT — pos=0, middle, beyond-end *)
    g_insert_mid  : STRING;
    g_insert_zero : STRING;
    g_insert_far  : STRING;

    (* DELETE — normal + no-op cases *)
    g_delete_mid  : STRING;
    g_delete_pos0 : STRING;
    g_delete_zero : STRING;
    g_delete_overrun : STRING;

    (* REPLACE — normal, replace at start, append *)
    g_replace_mid : STRING;
    g_replace_zero: STRING;
    g_replace_far : STRING;

    (* FIND *)
    g_find_yes    : INT;
    g_find_first  : INT;
    g_find_no     : INT;
    g_find_empty  : INT;

    (* Case conversion *)
    g_upper       : STRING;
    g_lower       : STRING;
    g_upper_alias : STRING;
    g_lower_alias : STRING;

    (* Trim *)
    g_trim        : STRING;
    g_ltrim       : STRING;
    g_rtrim       : STRING;

    (* Numeric → STRING *)
    g_int_to_s    : STRING;
    g_dint_to_s   : STRING;
    g_neg_to_s    : STRING;
    g_real_to_s   : STRING;
    g_real_int_s  : STRING;
    g_bool_t_to_s : STRING;
    g_bool_f_to_s : STRING;
    g_to_string_i : STRING;
    g_to_string_b : STRING;

    (* STRING → numeric *)
    g_s_to_int    : INT;
    g_s_to_int_neg: INT;
    g_s_to_real   : REAL;
    g_s_to_bool_t : INT;
    g_s_to_bool_1 : INT;
    g_s_to_bool_f : INT;
    g_s_to_int_bad: INT;

    (* Round-trip *)
    g_roundtrip_int : INT;
END_VAR

PROGRAM Main
VAR
    s         : STRING := 'hello';
    abc       : STRING := 'abcdef';
    spaces    : STRING := '  spaced  ';
    foo       : STRING := 'foo';
    bar       : STRING := 'bar';
    empty     : STRING := '';
    haystack  : STRING := 'rust-plc rocks';
    needle1   : STRING := 'plc';
    needle2   : STRING := 'X';
    n_int     : INT := 42;
    n_dint    : DINT := 1234567;
    n_neg     : INT := -7;
    n_real    : REAL := 3.5;
    n_real_i  : REAL := 1.0;
    s_num     : STRING := '123';
    s_neg_num : STRING := '-99';
    s_real    : STRING := '2.5';
    s_true    : STRING := 'TRUE';
    s_one     : STRING := '1';
    s_false   : STRING := 'false';
    s_bad     : STRING := 'banana';
    rt_text   : STRING;
END_VAR
    (* ── LEN ──────────────────────────────────────────────────────── *)
    g_len_hello := LEN(IN := s);                          (* 5 *)
    g_len_empty := LEN(IN := empty);                      (* 0 *)

    (* ── LEFT / RIGHT ─────────────────────────────────────────────── *)
    g_left_3     := LEFT(STR := abc, SIZE := 3);          (* 'abc' *)
    g_left_zero  := LEFT(STR := abc, SIZE := 0);          (* '' *)
    g_left_huge  := LEFT(STR := abc, SIZE := 100);        (* 'abcdef' *)
    g_left_neg   := LEFT(STR := abc, SIZE := -5);         (* '' *)
    g_right_3    := RIGHT(STR := abc, SIZE := 3);         (* 'def' *)
    g_right_zero := RIGHT(STR := abc, SIZE := 0);         (* '' *)
    g_right_huge := RIGHT(STR := abc, SIZE := 100);       (* 'abcdef' *)

    (* ── MID — 1-indexed, clamped ─────────────────────────────────── *)
    g_mid_mid     := MID(STR := abc, LEN := 3, POS := 2); (* 'bcd' *)
    g_mid_start   := MID(STR := abc, LEN := 2, POS := 1); (* 'ab' *)
    g_mid_end     := MID(STR := abc, LEN := 2, POS := 5); (* 'ef' *)
    g_mid_overrun := MID(STR := abc, LEN := 10, POS := 4);(* 'def' *)
    g_mid_pos0    := MID(STR := abc, LEN := 3, POS := 0); (* '' *)
    g_mid_negpos  := MID(STR := abc, LEN := 3, POS := -1);(* '' *)
    g_mid_zerolen := MID(STR := abc, LEN := 0, POS := 2); (* '' *)

    (* ── CONCAT ───────────────────────────────────────────────────── *)
    g_concat       := CONCAT(STR1 := foo, STR2 := bar);   (* 'foobar' *)
    g_concat_empty := CONCAT(STR1 := empty, STR2 := foo); (* 'foo' *)

    (* ── INSERT ───────────────────────────────────────────────────── *)
    g_insert_mid  := INSERT(STR1 := 'abef', STR2 := 'cd', POS := 2);  (* 'abcdef' *)
    g_insert_zero := INSERT(STR1 := abc, STR2 := 'XYZ', POS := 0);    (* 'XYZabcdef' *)
    g_insert_far  := INSERT(STR1 := abc, STR2 := 'XYZ', POS := 100);  (* 'abcdefXYZ' *)

    (* ── DELETE ───────────────────────────────────────────────────── *)
    g_delete_mid     := DELETE(STR := abc, LEN := 2, POS := 3);  (* 'abef' *)
    g_delete_pos0    := DELETE(STR := abc, LEN := 2, POS := 0);  (* 'abcdef' (no-op) *)
    g_delete_zero    := DELETE(STR := abc, LEN := 0, POS := 2);  (* 'abcdef' (no-op) *)
    g_delete_overrun := DELETE(STR := abc, LEN := 100, POS := 3);(* 'ab' *)

    (* ── REPLACE ──────────────────────────────────────────────────── *)
    g_replace_mid  := REPLACE(STR1 := abc, STR2 := 'XY', LEN := 3, POS := 2); (* 'aXYef' *)
    g_replace_zero := REPLACE(STR1 := abc, STR2 := 'XY', LEN := 2, POS := 0); (* 'XYcdef' (insert at start, drop 2) *)
    g_replace_far  := REPLACE(STR1 := abc, STR2 := 'XY', LEN := 1, POS := 100); (* 'abcdefXY' *)

    (* ── FIND (1-based, 0 = not found) ────────────────────────────── *)
    g_find_yes   := FIND(STR1 := haystack, STR2 := needle1);  (* 6 *)
    g_find_first := FIND(STR1 := 'aaa', STR2 := 'a');         (* 1 *)
    g_find_no    := FIND(STR1 := haystack, STR2 := needle2);  (* 0 *)
    g_find_empty := FIND(STR1 := haystack, STR2 := empty);    (* 0 *)

    (* ── Case ─────────────────────────────────────────────────────── *)
    g_upper       := TO_UPPER(IN := s);                    (* 'HELLO' *)
    g_lower       := TO_LOWER(IN := 'WORLD');              (* 'world' *)
    g_upper_alias := UPPER_CASE(IN := 'mixed');            (* 'MIXED' *)
    g_lower_alias := LOWER_CASE(IN := 'MIXED');            (* 'mixed' *)

    (* ── Trim ─────────────────────────────────────────────────────── *)
    g_trim  := TRIM(IN := spaces);                         (* 'spaced' *)
    g_ltrim := LTRIM(IN := spaces);                        (* 'spaced  ' *)
    g_rtrim := RTRIM(IN := spaces);                        (* '  spaced' *)

    (* ── Numeric → STRING ─────────────────────────────────────────── *)
    g_int_to_s    := INT_TO_STRING(IN := n_int);           (* '42' *)
    g_dint_to_s   := DINT_TO_STRING(IN := n_dint);         (* '1234567' *)
    g_neg_to_s    := INT_TO_STRING(IN := n_neg);           (* '-7' *)
    g_real_to_s   := REAL_TO_STRING(IN := n_real);         (* '3.5' *)
    g_real_int_s  := REAL_TO_STRING(IN := n_real_i);       (* '1.0' *)
    g_bool_t_to_s := BOOL_TO_STRING(IN := TRUE);           (* 'TRUE' *)
    g_bool_f_to_s := BOOL_TO_STRING(IN := FALSE);          (* 'FALSE' *)
    g_to_string_i := TO_STRING(IN := 99);                  (* '99' *)
    g_to_string_b := TO_STRING(IN := TRUE);                (* 'TRUE' *)

    (* ── STRING → numeric ─────────────────────────────────────────── *)
    g_s_to_int     := STRING_TO_INT(IN := s_num);          (* 123 *)
    g_s_to_int_neg := STRING_TO_INT(IN := s_neg_num);      (* -99 *)
    g_s_to_real    := STRING_TO_REAL(IN := s_real);        (* 2.5 *)
    g_s_to_bool_t  := BOOL_TO_INT(IN := STRING_TO_BOOL(IN := s_true));  (* 1 *)
    g_s_to_bool_1  := BOOL_TO_INT(IN := STRING_TO_BOOL(IN := s_one));   (* 1 *)
    g_s_to_bool_f  := BOOL_TO_INT(IN := STRING_TO_BOOL(IN := s_false)); (* 0 *)
    g_s_to_int_bad := STRING_TO_INT(IN := s_bad);          (* 0 (parse fail) *)

    (* ── Round-trip: INT → STRING → INT ───────────────────────────── *)
    rt_text         := INT_TO_STRING(IN := 17);
    g_roundtrip_int := STRING_TO_INT(IN := rt_text);       (* 17 *)
END_PROGRAM
